LIN {X 0,Y 488.67,Z 344.234,A -85,B 0,C 180,E1 -6456.253,E2 -6456.253} C_VEL
LIN {X 0,Y 488.747,Z 344.224,A -85,B 0,C 180,E1 -6459.176,E2 -6459.176} C_VEL
LIN {X 0,Y 488.748,Z 344.228,A -85,B 0,C 180,E1 -6461.632,E2 -6461.632} C_VEL
LIN {X 0,Y 488.762,Z 344.223,A -85,B 0,C 180,E1 -6465,E2 -6465} C_VEL
LIN {X 0,Y 488.806,Z 344.211,A -85,B 0,C 180,E1 -6468.387,E2 -6468.387} C_VEL
LIN {X 0,Y 488.786,Z 344.226,A -85,B 0,C 180,E1 -6471.733,E2 -6471.733} C_VEL
LIN {X 0,Y 488.853,Z 344.206,A -85,B 0,C 180,E1 -6474.224,E2 -6474.224} C_VEL
LIN {X 0,Y 488.953,Z 344.207,A -85,B 0,C 180,E1 -6477.529,E2 -6477.529} C_VEL
LIN {X 0,Y 488.97,Z 344.194,A -85,B 0,C 180,E1 -6480,E2 -6480} C_VEL
LIN {X 0,Y 488.956,Z 344.194,A -85,B 0,C 180,E1 -6482.471,E2 -6482.471} C_VEL
LIN {X 0,Y 488.842,Z 344.213,A -85,B 0,C 180,E1 -6485.776,E2 -6485.776} C_VEL
LIN {X 0,Y 488.787,Z 344.212,A -85,B 0,C 180,E1 -6488.267,E2 -6488.267} C_VEL
LIN {X 0,Y 488.806,Z 344.219,A -85,B 0,C 180,E1 -6491.612,E2 -6491.612} C_VEL
LIN {X 0,Y 488.762,Z 344.22,A -85,B 0,C 180,E1 -6495,E2 -6495} C_VEL
LIN {X 0,Y 488.747,Z 344.223,A -85,B 0,C 180,E1 -6498.442,E2 -6498.442} C_VEL
LIN {X 0,Y 488.707,Z 344.231,A -85,B 0,C 180,E1 -6501.071,E2 -6501.071} C_VEL
LIN {X 0,Y 488.684,Z 344.231,A -85,B 0,C 180,E1 -6503.746,E2 -6503.746} C_VEL
LIN {X 0,Y 488.792,Z 344.223,A -85,B 0,C 180,E1 -6506.944,E2 -6506.944} C_VEL
LIN {X 0,Y 488.71,Z 344.225,A -85,B 0,C 180,E1 -6510.363,E2 -6510.363} C_VEL
LIN {X 0,Y 488.734,Z 344.226,A -85,B 0,C 180,E1 -6513.484,E2 -6513.484} C_VEL
LIN {X 0,Y 488.682,Z 344.235,A -85,B 0,C 180,E1 -6516.354,E2 -6516.354} C_VEL
LIN {X 0,Y 488.701,Z 344.217,A -85,B 0,C 180,E1 -6519.254,E2 -6519.254} C_VEL
LIN {X 0,Y 488.709,Z 344.228,A -85,B 0,C 180,E1 -6521.6,E2 -6521.6} C_VEL
LIN {X 0,Y 488.712,Z 344.234,A -85,B 0,C 180,E1 -6524.801,E2 -6524.801} C_VEL
LIN {X 0,Y 488.692,Z 344.227,A -85,B 0,C 180,E1 -6527.475,E2 -6527.475} C_VEL
LIN {X 0,Y 488.733,Z 344.229,A -85,B 0,C 180,E1 -6529.677,E2 -6529.677} C_VEL
LIN {X 0,Y 488.68,Z 344.241,A -85,B 0,C 180,E1 -6532.841,E2 -6532.841} C_VEL
LIN {X 0,Y 488.73,Z 344.231,A -85,B 0,C 180,E1 -6535.887,E2 -6535.887} C_VEL
LIN {X 0,Y 488.692,Z 344.238,A -85,B 0,C 180,E1 -6538.82,E2 -6538.82} C_VEL
LIN {X 0,Y 488.769,Z 344.487,A -85,B 0,C 180,E1 -6540.052,E2 -6540.052} C_VEL
LIN {X 0,Y 493.274,Z 361.433,A -85,B 0,C 180,E1 -6542.558,E2 -6542.558} C_VEL
LIN {X 0,Y 493.811,Z 363.917,A -85,B 0,C 180,E1 -6542.907,E2 -6542.907} C_VEL
LIN {X 0,Y 492.75,Z 385.348,A -85,B 0,C 180,E1 -6545.568,E2 -6545.568} C_VEL
LIN {X 0,Y 492.176,Z 397.96,A -85,B 0,C 180,E1 -6547.086,E2 -6547.086} C_VEL
LIN {X 0,Y 493.705,Z 407.128,A -85,B 0,C 180,E1 -6547.34,E2 -6547.34} C_VEL
LIN {X 0,Y 495.118,Z 416.237,A -85,B 0,C 180,E1 -6547.557,E2 -6547.557} C_VEL
LIN {X 0,Y 493.738,Z 536.271,A -85,B 0,C 180,E1 -6549.427,E2 -6549.427} C_VEL
LIN {X 0,Y 493.419,Z 566.389,A -85,B 0,C 180,E1 -6549.902,E2 -6549.902} C_VEL
LIN {X 0,Y 493.068,Z 581.521,A -85,B 0,C 180,E1 -6550.306,E2 -6550.306} C_VEL
LIN {X 0,Y 492.614,Z 595.743,A -85,B 0,C 180,E1 -6550.844,E2 -6550.844} C_VEL
LIN {X 0,Y 491.977,Z 610.35,A -85,B 0,C 180,E1 -6551.575,E2 -6551.575} C_VEL
LIN {X 0,Y 491.358,Z 623.614,A -85,B 0,C 180,E1 -6552.413,E2 -6552.413} C_VEL
LIN {X 0,Y 490.716,Z 636.907,A -85,B 0,C 180,E1 -6553.447,E2 -6553.447} C_VEL
LIN {X 0,Y 490.068,Z 649.271,A -85,B 0,C 180,E1 -6554.615,E2 -6554.615} C_VEL
LIN {X 0,Y 489.488,Z 660.375,A -85,B 0,C 180,E1 -6555.872,E2 -6555.872} C_VEL
LIN {X 0,Y 488.978,Z 671.128,A -85,B 0,C 180,E1 -6557.339,E2 -6557.339} C_VEL
LIN {X 0,Y 488.576,Z 680.063,A -85,B 0,C 180,E1 -6558.803,E2 -6558.803} C_VEL
LIN {X 0,Y 488.296,Z 686.584,A -85,B 0,C 180,E1 -6560.054,E2 -6560.054} C_VEL
LIN {X 0,Y 488.131,Z 693.802,A -85,B 0,C 180,E1 -6561.722,E2 -6561.722} C_VEL
LIN {X 0,Y 487.997,Z 699.465,A -85,B 0,C 180,E1 -6563.384,E2 -6563.384} C_VEL
LIN {X 0,Y 487.928,Z 703.738,A -85,B 0,C 180,E1 -6565.042,E2 -6565.042} C_VEL
LIN {X 0,Y 487.946,Z 706.729,A -85,B 0,C 180,E1 -6566.697,E2 -6566.697} C_VEL
LIN {X 0,Y 487.889,Z 708.505,A -85,B 0,C 180,E1 -6568.349,E2 -6568.349} C_VEL
LIN {X 0,Y 487.816,Z 709.096,A -85,B 0,C 180,E1 -6570,E2 -6570} C_VEL
LIN {X 0,Y 487.89,Z 708.466,A -85,B 0,C 180,E1 -6571.651,E2 -6571.651} C_VEL
LIN {X 0,Y 487.947,Z 706.652,A -85,B 0,C 180,E1 -6573.303,E2 -6573.303} C_VEL
LIN {X 0,Y 487.927,Z 703.612,A -85,B 0,C 180,E1 -6574.958,E2 -6574.958} C_VEL
LIN {X 0,Y 487.992,Z 699.278,A -85,B 0,C 180,E1 -6576.616,E2 -6576.616} C_VEL
LIN {X 0,Y 488.131,Z 693.56,A -85,B 0,C 180,E1 -6578.278,E2 -6578.278} C_VEL
LIN {X 0,Y 488.294,Z 686.458,A -85,B 0,C 180,E1 -6579.946,E2 -6579.946} C_VEL
LIN {X 0,Y 488.641,Z 678.867,A -85,B 0,C 180,E1 -6581.406,E2 -6581.406} C_VEL
LIN {X 0,Y 489.055,Z 669.708,A -85,B 0,C 180,E1 -6582.87,E2 -6582.87} C_VEL
LIN {X 0,Y 489.498,Z 660.375,A -85,B 0,C 180,E1 -6584.128,E2 -6584.128} C_VEL
LIN {X 0,Y 490.044,Z 649.264,A -85,B 0,C 180,E1 -6585.386,E2 -6585.386} C_VEL
LIN {X 0,Y 490.741,Z 636.855,A -85,B 0,C 180,E1 -6586.556,E2 -6586.556} C_VEL
LIN {X 0,Y 491.377,Z 623.612,A -85,B 0,C 180,E1 -6587.587,E2 -6587.587} C_VEL
LIN {X 0,Y 491.994,Z 610.353,A -85,B 0,C 180,E1 -6588.424,E2 -6588.424} C_VEL
LIN {X 0,Y 492.62,Z 595.727,A -85,B 0,C 180,E1 -6589.156,E2 -6589.156} C_VEL
LIN {X 0,Y 493.109,Z 580.58,A -85,B 0,C 180,E1 -6589.725,E2 -6589.725} C_VEL
LIN {X 0,Y 493.458,Z 565.175,A -85,B 0,C 180,E1 -6590.123,E2 -6590.123} C_VEL
LIN {X 0,Y 494.855,Z 418.053,A -85,B 0,C 180,E1 -6592.352,E2 -6592.352} C_VEL
LIN {X 0,Y 494.694,Z 413.968,A -85,B 0,C 180,E1 -6592.433,E2 -6592.433} C_VEL
LIN {X 0,Y 492.106,Z 398.162,A -85,B 0,C 180,E1 -6592.861,E2 -6592.861} C_VEL
LIN {X 0,Y 493.384,Z 375.124,A -85,B 0,C 180,E1 -6595.737,E2 -6595.737} C_VEL
LIN {X 0,Y 494.102,Z 364.814,A -85,B 0,C 180,E1 -6597.075,E2 -6597.075} C_VEL
LIN {X 0,Y 491.36,Z 353.308,A -85,B 0,C 180,E1 -6598.888,E2 -6598.888} C_VEL
LIN {X 0,Y 488.742,Z 344.352,A -85,B 0,C 180,E1 -6600.478,E2 -6600.478} C_VEL
LIN {X 0,Y 488.736,Z 344.232,A -85,B 0,C 180,E1 -6603.484,E2 -6603.484} C_VEL
LIN {X 0,Y 488.685,Z 344.239,A -85,B 0,C 180,E1 -6606.355,E2 -6606.355} C_VEL
LIN {X 0,Y 488.702,Z 344.238,A -85,B 0,C 180,E1 -6609.254,E2 -6609.254} C_VEL
LIN {X 0,Y 488.707,Z 344.233,A -85,B 0,C 180,E1 -6611.6,E2 -6611.6} C_VEL
LIN {X 0,Y 488.702,Z 344.239,A -85,B 0,C 180,E1 -6614.803,E2 -6614.803} C_VEL
LIN {X 0,Y 488.689,Z 344.236,A -85,B 0,C 180,E1 -6617.474,E2 -6617.474} C_VEL
LIN {X 0,Y 488.701,Z 344.238,A -85,B 0,C 180,E1 -6620.746,E2 -6620.746} C_VEL
LIN {X 0,Y 488.67,Z 344.241,A -85,B 0,C 180,E1 -6623.867,E2 -6623.867} C_VEL
LIN {X 0,Y 488.737,Z 344.233,A -85,B 0,C 180,E1 -6626.877,E2 -6626.877} C_VEL
LIN {X 0,Y 488.719,Z 344.236,A -85,B 0,C 180,E1 -6629.78,E2 -6629.78} C_VEL
LIN {X 0,Y 488.736,Z 344.505,A -85,B 0,C 180,E1 -6631.148,E2 -6631.148} C_VEL
LIN {X 0,Y 491.865,Z 356.433,A -85,B 0,C 180,E1 -6633.48,E2 -6633.48} C_VEL
LIN {X 0,Y 493.058,Z 363.175,A -85,B 0,C 180,E1 -6634.684,E2 -6634.684} C_VEL
LIN {X 0,Y 491.663,Z 386.383,A -85,B 0,C 180,E1 -6638.3,E2 -6638.3} C_VEL
LIN {X 0,Y 491.166,Z 398.04,A -85,B 0,C 180,E1 -6640.038,E2 -6640.038} C_VEL
LIN {X 0,Y 494.175,Z 414.23,A -85,B 0,C 180,E1 -6640.519,E2 -6640.519} C_VEL
LIN {X 0,Y 492.63,Z 511.877,A -85,B 0,C 180,E1 -6642.219,E2 -6642.219} C_VEL
LIN {X 0,Y 492.189,Z 540.322,A -85,B 0,C 180,E1 -6642.728,E2 -6642.728} C_VEL
LIN {X 0,Y 491.852,Z 554.764,A -85,B 0,C 180,E1 -6643.155,E2 -6643.155} C_VEL
LIN {X 0,Y 491.483,Z 569.057,A -85,B 0,C 180,E1 -6643.756,E2 -6643.756} C_VEL
LIN {X 0,Y 491.035,Z 581.402,A -85,B 0,C 180,E1 -6644.433,E2 -6644.433} C_VEL
LIN {X 0,Y 490.524,Z 593.611,A -85,B 0,C 180,E1 -6645.267,E2 -6645.267} C_VEL
LIN {X 0,Y 490.005,Z 605.948,A -85,B 0,C 180,E1 -6646.311,E2 -6646.311} C_VEL
LIN {X 0,Y 489.55,Z 616.291,A -85,B 0,C 180,E1 -6647.375,E2 -6647.375} C_VEL
LIN {X 0,Y 489.153,Z 626.192,A -85,B 0,C 180,E1 -6648.606,E2 -6648.606} C_VEL
LIN {X 0,Y 488.76,Z 634.535,A -85,B 0,C 180,E1 -6649.855,E2 -6649.855} C_VEL
LIN {X 0,Y 488.47,Z 642.486,A -85,B 0,C 180,E1 -6651.311,E2 -6651.311} C_VEL
LIN {X 0,Y 488.253,Z 648.047,A -85,B 0,C 180,E1 -6652.557,E2 -6652.557} C_VEL
LIN {X 0,Y 488.163,Z 653.848,A -85,B 0,C 180,E1 -6654.216,E2 -6654.216} C_VEL
LIN {X 0,Y 487.974,Z 656.147,A -85,B 0,C 180,E1 -6655.043,E2 -6655.043} C_VEL
LIN {X 0,Y 488.064,Z 658.053,A -85,B 0,C 180,E1 -6655.871,E2 -6655.871} C_VEL
LIN {X 0,Y 487.987,Z 660.799,A -85,B 0,C 180,E1 -6657.524,E2 -6657.524} C_VEL
LIN {X 0,Y 487.831,Z 662.169,A -85,B 0,C 180,E1 -6659.175,E2 -6659.175} C_VEL
LIN {X 0,Y 487.831,Z 662.181,A -85,B 0,C 180,E1 -6660.826,E2 -6660.826} C_VEL
LIN {X 0,Y 487.987,Z 660.829,A -85,B 0,C 180,E1 -6662.476,E2 -6662.476} C_VEL
LIN {X 0,Y 488.043,Z 658.097,A -85,B 0,C 180,E1 -6664.129,E2 -6664.129} C_VEL
LIN {X 0,Y 488.06,Z 655.112,A -85,B 0,C 180,E1 -6665.371,E2 -6665.371} C_VEL
LIN {X 0,Y 488.144,Z 651.07,A -85,B 0,C 180,E1 -6666.663,E2 -6666.663} C_VEL
LIN {X 0,Y 488.36,Z 644.627,A -85,B 0,C 180,E1 -6668.274,E2 -6668.274} C_VEL
LIN {X 0,Y 488.647,Z 637.248,A -85,B 0,C 180,E1 -6669.73,E2 -6669.73} C_VEL
LIN {X 0,Y 489.05,Z 628.073,A -85,B 0,C 180,E1 -6671.187,E2 -6671.187} C_VEL
LIN {X 0,Y 489.464,Z 618.122,A -85,B 0,C 180,E1 -6672.476,E2 -6672.476} C_VEL
LIN {X 0,Y 489.886,Z 607.773,A -85,B 0,C 180,E1 -6673.587,E2 -6673.587} C_VEL
LIN {X 0,Y 490.398,Z 595.975,A -85,B 0,C 180,E1 -6674.631,E2 -6674.631} C_VEL
LIN {X 0,Y 490.984,Z 582.874,A -85,B 0,C 180,E1 -6675.569,E2 -6675.569} C_VEL
LIN {X 0,Y 491.461,Z 570.021,A -85,B 0,C 180,E1 -6676.299,E2 -6676.299} C_VEL
LIN {X 0,Y 491.859,Z 555.768,A -85,B 0,C 180,E1 -6676.918,E2 -6676.918} C_VEL
LIN {X 0,Y 492.294,Z 541.273,A -85,B 0,C 180,E1 -6677.357,E2 -6677.357} C_VEL
LIN {X 0,Y 492.476,Z 525.847,A -85,B 0,C 180,E1 -6677.653,E2 -6677.653} C_VEL
LIN {X 0,Y 493.822,Z 414.339,A -85,B 0,C 180,E1 -6679.448,E2 -6679.448} C_VEL
LIN {X 0,Y 490.808,Z 397.758,A -85,B 0,C 180,E1 -6679.875,E2 -6679.875} C_VEL
LIN {X 0,Y 491.591,Z 378.455,A -85,B 0,C 180,E1 -6682.706,E2 -6682.706} C_VEL
LIN {X 0,Y 492.374,Z 360.916,A -85,B 0,C 180,E1 -6685.354,E2 -6685.354} C_VEL
LIN {X 0,Y 490.258,Z 350.903,A -85,B 0,C 180,E1 -6687.034,E2 -6687.034} C_VEL
LIN {X 0,Y 488.753,Z 344.554,A -85,B 0,C 180,E1 -6688.153,E2 -6688.153} C_VEL
LIN {X 0,Y 488.695,Z 344.246,A -85,B 0,C 180,E1 -6688.332,E2 -6688.332} C_VEL
LIN {X 0,Y 488.659,Z 344.24,A -85,B 0,C 180,E1 -6691.182,E2 -6691.182} C_VEL
LIN {X 0,Y 488.703,Z 344.239,A -85,B 0,C 180,E1 -6694.115,E2 -6694.115} C_VEL
LIN {X 0,Y 488.646,Z 344.24,A -85,B 0,C 180,E1 -6697.162,E2 -6697.162} C_VEL
LIN {X 0,Y 488.668,Z 344.24,A -85,B 0,C 180,E1 -6700.33,E2 -6700.33} C_VEL
LIN {X 0,Y 488.658,Z 344.232,A -85,B 0,C 180,E1 -6703.562,E2 -6703.562} C_VEL
LIN {X 0,Y 488.027,Z 344.322,A -85,B 0,C 180,E1 -6704.249,E2 -6704.249} C_VEL
LIN {X 0,Y 485.175,Z 344.673,A -85,B 0,C 180,E1 -6705.366,E2 -6705.366} C_VEL
LIN {X 0,Y 482.736,Z 344.972,A -85,B 0,C 180,E1 -6706.266,E2 -6706.266} C_VEL
LIN {X 0,Y 481.682,Z 345.099,A -85,B 0,C 180,E1 -6706.962,E2 -6706.962} C_VEL
LIN {X 0,Y 481.595,Z 345.11,A -85,B 0,C 180,E1 -6707.197,E2 -6707.197} C_VEL
LIN {X 0,Y 481.628,Z 345.113,A -85,B 0,C 180,E1 -6710.055,E2 -6710.055} C_VEL
LIN {X 0,Y 481.603,Z 345.114,A -85,B 0,C 180,E1 -6713.251,E2 -6713.251} C_VEL
LIN {X 0,Y 481.671,Z 345.113,A -85,B 0,C 180,E1 -6716.327,E2 -6716.327} C_VEL
LIN {X 0,Y 481.632,Z 345.309,A -85,B 0,C 180,E1 -6719.478,E2 -6719.478} C_VEL
LIN {X 0,Y 485.46,Z 360.506,A -85,B 0,C 180,E1 -6721.798,E2 -6721.798} C_VEL
LIN {X 0,Y 486.304,Z 365.031,A -85,B 0,C 180,E1 -6722.454,E2 -6722.454} C_VEL
LIN {X 0,Y 485.411,Z 387.512,A -85,B 0,C 180,E1 -6725.385,E2 -6725.385} C_VEL
LIN {X 0,Y 485.132,Z 397.848,A -85,B 0,C 180,E1 -6726.645,E2 -6726.645} C_VEL
LIN {X 0,Y 488.991,Z 418.099,A -85,B 0,C 180,E1 -6727.166,E2 -6727.166} C_VEL
LIN {X 0,Y 487.489,Z 565.061,A -85,B 0,C 180,E1 -6729.407,E2 -6729.407} C_VEL
LIN {X 0,Y 487.064,Z 580.106,A -85,B 0,C 180,E1 -6729.794,E2 -6729.794} C_VEL
LIN {X 0,Y 486.479,Z 595.122,A -85,B 0,C 180,E1 -6730.351,E2 -6730.351} C_VEL
LIN {X 0,Y 485.866,Z 608.495,A -85,B 0,C 180,E1 -6731.006,E2 -6731.006} C_VEL
LIN {X 0,Y 485.213,Z 622.242,A -85,B 0,C 180,E1 -6731.855,E2 -6731.855} C_VEL
LIN {X 0,Y 484.433,Z 634.862,A -85,B 0,C 180,E1 -6732.807,E2 -6732.807} C_VEL
LIN {X 0,Y 483.707,Z 647.615,A -85,B 0,C 180,E1 -6733.975,E2 -6733.975} C_VEL
LIN {X 0,Y 483.081,Z 657.437,A -85,B 0,C 180,E1 -6735.035,E2 -6735.035} C_VEL
LIN {X 0,Y 482.49,Z 667.455,A -85,B 0,C 180,E1 -6736.308,E2 -6736.308} C_VEL
LIN {X 0,Y 481.889,Z 677.81,A -85,B 0,C 180,E1 -6737.888,E2 -6737.888} C_VEL
LIN {X 0,Y 481.597,Z 685.38,A -85,B 0,C 180,E1 -6739.277,E2 -6739.277} C_VEL
LIN {X 0,Y 481.239,Z 692.115,A -85,B 0,C 180,E1 -6740.756,E2 -6740.756} C_VEL
LIN {X 0,Y 481.016,Z 698.355,A -85,B 0,C 180,E1 -6742.444,E2 -6742.444} C_VEL
LIN {X 0,Y 480.915,Z 703.186,A -85,B 0,C 180,E1 -6744.128,E2 -6744.128} C_VEL
LIN {X 0,Y 480.796,Z 706.733,A -85,B 0,C 180,E1 -6745.809,E2 -6745.809} C_VEL
LIN {X 0,Y 480.8,Z 709.075,A -85,B 0,C 180,E1 -6747.487,E2 -6747.487} C_VEL
LIN {X 0,Y 480.757,Z 710.268,A -85,B 0,C 180,E1 -6749.162,E2 -6749.162} C_VEL
LIN {X 0,Y 480.757,Z 710.285,A -85,B 0,C 180,E1 -6750.838,E2 -6750.838} C_VEL
LIN {X 0,Y 480.8,Z 709.156,A -85,B 0,C 180,E1 -6752.513,E2 -6752.513} C_VEL
LIN {X 0,Y 480.796,Z 706.883,A -85,B 0,C 180,E1 -6754.191,E2 -6754.191} C_VEL
LIN {X 0,Y 480.921,Z 703.413,A -85,B 0,C 180,E1 -6755.871,E2 -6755.871} C_VEL
LIN {X 0,Y 481.009,Z 698.658,A -85,B 0,C 180,E1 -6757.556,E2 -6757.556} C_VEL
LIN {X 0,Y 481.219,Z 692.491,A -85,B 0,C 180,E1 -6759.245,E2 -6759.245} C_VEL
LIN {X 0,Y 481.617,Z 684.74,A -85,B 0,C 180,E1 -6760.935,E2 -6760.935} C_VEL
LIN {X 0,Y 482.001,Z 676.224,A -85,B 0,C 180,E1 -6762.461,E2 -6762.461} C_VEL
LIN {X 0,Y 482.563,Z 666.53,A -85,B 0,C 180,E1 -6763.904,E2 -6763.904} C_VEL
LIN {X 0,Y 483.131,Z 656.375,A -85,B 0,C 180,E1 -6765.179,E2 -6765.179} C_VEL
LIN {X 0,Y 483.861,Z 644.214,A -85,B 0,C 180,E1 -6766.454,E2 -6766.454} C_VEL
LIN {X 0,Y 484.626,Z 632.086,A -85,B 0,C 180,E1 -6767.512,E2 -6767.512} C_VEL
LIN {X 0,Y 485.389,Z 618.859,A -85,B 0,C 180,E1 -6768.465,E2 -6768.465} C_VEL
LIN {X 0,Y 486.055,Z 605.273,A -85,B 0,C 180,E1 -6769.26,E2 -6769.26} C_VEL
LIN {X 0,Y 486.718,Z 589.87,A -85,B 0,C 180,E1 -6769.958,E2 -6769.958} C_VEL
LIN {X 0,Y 487.207,Z 575.123,A -85,B 0,C 180,E1 -6770.448,E2 -6770.448} C_VEL
LIN {X 0,Y 487.572,Z 559.443,A -85,B 0,C 180,E1 -6770.79,E2 -6770.79} C_VEL
LIN {X 0,Y 488.93,Z 417.561,A -85,B 0,C 180,E1 -6772.936,E2 -6772.936} C_VEL
LIN {X 0,Y 485.145,Z 397.66,A -85,B 0,C 180,E1 -6773.458,E2 -6773.458} C_VEL
LIN {X 0,Y 485.658,Z 381.364,A -85,B 0,C 180,E1 -6775.5,E2 -6775.5} C_VEL
LIN {X 0,Y 486.267,Z 364.634,A -85,B 0,C 180,E1 -6777.698,E2 -6777.698} C_VEL
LIN {X 0,Y 483.266,Z 351.613,A -85,B 0,C 180,E1 -6779.634,E2 -6779.634} C_VEL
LIN {X 0,Y 481.645,Z 345.259,A -85,B 0,C 180,E1 -6780.631,E2 -6780.631} C_VEL
LIN {X 0,Y 481.649,Z 345.109,A -85,B 0,C 180,E1 -6783.724,E2 -6783.724} C_VEL
LIN {X 0,Y 481.602,Z 345.118,A -85,B 0,C 180,E1 -6786.749,E2 -6786.749} C_VEL
LIN {X 0,Y 481.627,Z 345.11,A -85,B 0,C 180,E1 -6789.945,E2 -6789.945} C_VEL
LIN {X 0,Y 481.618,Z 345.115,A -85,B 0,C 180,E1 -6793.302,E2 -6793.302} C_VEL
LIN {X 0,Y 481.652,Z 345.113,A -85,B 0,C 180,E1 -6795.642,E2 -6795.642} C_VEL
LIN {X 0,Y 481.62,Z 345.115,A -85,B 0,C 180,E1 -6798.954,E2 -6798.954} C_VEL
LIN {X 0,Y 481.633,Z 345.119,A -85,B 0,C 180,E1 -6801.996,E2 -6801.996} C_VEL
LIN {X 0,Y 481.68,Z 345.105,A -85,B 0,C 180,E1 -6805.317,E2 -6805.317} C_VEL
LIN {X 0,Y 481.643,Z 345.107,A -85,B 0,C 180,E1 -6808.311,E2 -6808.311} C_VEL
LIN {X 0,Y 481.673,Z 345.11,A -85,B 0,C 180,E1 -6811.217,E2 -6811.217} C_VEL
LIN {X 0,Y 481.643,Z 345.114,A -85,B 0,C 180,E1 -6814.039,E2 -6814.039} C_VEL
LIN {X 0,Y 481.675,Z 345.105,A -85,B 0,C 180,E1 -6816.812,E2 -6816.812} C_VEL
LIN {X 0,Y 481.696,Z 345.107,A -85,B 0,C 180,E1 -6819.503,E2 -6819.503} C_VEL
LIN {X 0,Y 481.689,Z 345.101,A -85,B 0,C 180,E1 -6822.158,E2 -6822.158} C_VEL
LIN {X 0,Y 481.743,Z 345.096,A -85,B 0,C 180,E1 -6824.776,E2 -6824.776} C_VEL
LIN {X 0,Y 481.752,Z 345.091,A -85,B 0,C 180,E1 -6828.215,E2 -6828.215} C_VEL
LIN {X 0,Y 481.74,Z 345.105,A -85,B 0,C 180,E1 -6831.611,E2 -6831.611} C_VEL
LIN {X 0,Y 481.814,Z 345.083,A -85,B 0,C 180,E1 -6834.139,E2 -6834.139} C_VEL
LIN {X 0,Y 481.919,Z 345.082,A -85,B 0,C 180,E1 -6837.492,E2 -6837.492} C_VEL
LIN {X 0,Y 481.941,Z 345.07,A -85,B 0,C 180,E1 -6840,E2 -6840} C_VEL
LIN {X 0,Y 481.922,Z 345.07,A -85,B 0,C 180,E1 -6842.507,E2 -6842.507} C_VEL
LIN {X 0,Y 481.801,Z 345.089,A -85,B 0,C 180,E1 -6845.861,E2 -6845.861} C_VEL
LIN {X 0,Y 481.741,Z 345.09,A -85,B 0,C 180,E1 -6848.389,E2 -6848.389} C_VEL
LIN {X 0,Y 481.752,Z 345.096,A -85,B 0,C 180,E1 -6851.785,E2 -6851.785} C_VEL
LIN {X 0,Y 481.743,Z 345.098,A -85,B 0,C 180,E1 -6855.224,E2 -6855.224} C_VEL
LIN {X 0,Y 481.709,Z 345.101,A -85,B 0,C 180,E1 -6858.722,E2 -6858.722} C_VEL
LIN {X 0,Y 481.647,Z 345.116,A -85,B 0,C 180,E1 -6861.395,E2 -6861.395} C_VEL
LIN {X 0,Y 481.67,Z 345.103,A -85,B 0,C 180,E1 -6864.113,E2 -6864.113} C_VEL
LIN {X 0,Y 481.747,Z 345.104,A -85,B 0,C 180,E1 -6867.139,E2 -6867.139} C_VEL
LIN {X 0,Y 481.679,Z 345.101,A -85,B 0,C 180,E1 -6869.741,E2 -6869.741} C_VEL
LIN {X 0,Y 481.672,Z 345.111,A -85,B 0,C 180,E1 -6872.674,E2 -6872.674} C_VEL
LIN {X 0,Y 481.637,Z 345.113,A -85,B 0,C 180,E1 -6875.709,E2 -6875.709} C_VEL
LIN {X 0,Y 481.671,Z 345.099,A -85,B 0,C 180,E1 -6878.859,E2 -6878.859} C_VEL
LIN {X 0,Y 481.654,Z 345.105,A -85,B 0,C 180,E1 -6881.913,E2 -6881.913} C_VEL
LIN {X 0,Y 481.66,Z 345.112,A -85,B 0,C 180,E1 -6884.457,E2 -6884.457} C_VEL
LIN {X 0,Y 481.648,Z 345.105,A -85,B 0,C 180,E1 -6887.839,E2 -6887.839} C_VEL
LIN {X 0,Y 481.681,Z 345.111,A -85,B 0,C 180,E1 -6890.651,E2 -6890.651} C_VEL
LIN {X 0,Y 481.627,Z 345.116,A -85,B 0,C 180,E1 -6893.376,E2 -6893.376} C_VEL
LIN {X 0,Y 481.71,Z 345.108,A -85,B 0,C 180,E1 -6896.33,E2 -6896.33} C_VEL
LIN {X 0,Y 481.72,Z 345.277,A -85,B 0,C 180,E1 -6899.69,E2 -6899.69} C_VEL
LIN {X 0,Y 486.112,Z 361.759,A -85,B 0,C 180,E1 -6902.185,E2 -6902.185} C_VEL
LIN {X 0,Y 486.996,Z 365.544,A -85,B 0,C 180,E1 -6902.729,E2 -6902.729} C_VEL
LIN {X 0,Y 486.309,Z 379.817,A -85,B 0,C 180,E1 -6904.536,E2 -6904.536} C_VEL
LIN {X 0,Y 485.379,Z 397.859,A -85,B 0,C 180,E1 -6906.761,E2 -6906.761} C_VEL
LIN {X 0,Y 486.072,Z 402.084,A -85,B 0,C 180,E1 -6906.908,E2 -6906.908} C_VEL
LIN {X 0,Y 488.492,Z 417.195,A -85,B 0,C 180,E1 -6907.274,E2 -6907.274} C_VEL
LIN {X 0,Y 487.464,Z 502.409,A -85,B 0,C 180,E1 -6908.624,E2 -6908.624} C_VEL
LIN {X 0,Y 486.823,Z 565.34,A -85,B 0,C 180,E1 -6909.59,E2 -6909.59} C_VEL
LIN {X 0,Y 486.403,Z 581.053,A -85,B 0,C 180,E1 -6910.004,E2 -6910.004} C_VEL
LIN {X 0,Y 485.904,Z 595.807,A -85,B 0,C 180,E1 -6910.569,E2 -6910.569} C_VEL
LIN {X 0,Y 485.218,Z 610.4,A -85,B 0,C 180,E1 -6911.309,E2 -6911.309} C_VEL
LIN {X 0,Y 484.563,Z 623.657,A -85,B 0,C 180,E1 -6912.158,E2 -6912.158} C_VEL
LIN {X 0,Y 483.853,Z 637.104,A -85,B 0,C 180,E1 -6913.22,E2 -6913.22} C_VEL
LIN {X 0,Y 483.156,Z 649.303,A -85,B 0,C 180,E1 -6914.389,E2 -6914.389} C_VEL
LIN {X 0,Y 482.537,Z 660.403,A -85,B 0,C 180,E1 -6915.665,E2 -6915.665} C_VEL
LIN {X 0,Y 481.997,Z 671.152,A -85,B 0,C 180,E1 -6917.152,E2 -6917.152} C_VEL
LIN {X 0,Y 481.565,Z 680.074,A -85,B 0,C 180,E1 -6918.637,E2 -6918.637} C_VEL
LIN {X 0,Y 481.257,Z 686.473,A -85,B 0,C 180,E1 -6919.907,E2 -6919.907} C_VEL
LIN {X 0,Y 481.057,Z 693.547,A -85,B 0,C 180,E1 -6921.599,E2 -6921.599} C_VEL
LIN {X 0,Y 480.908,Z 699.113,A -85,B 0,C 180,E1 -6923.286,E2 -6923.286} C_VEL
LIN {X 0,Y 480.854,Z 703.387,A -85,B 0,C 180,E1 -6924.969,E2 -6924.969} C_VEL
LIN {X 0,Y 480.87,Z 706.389,A -85,B 0,C 180,E1 -6926.649,E2 -6926.649} C_VEL
LIN {X 0,Y 480.82,Z 708.17,A -85,B 0,C 180,E1 -6928.325,E2 -6928.325} C_VEL
LIN {X 0,Y 480.74,Z 708.76,A -85,B 0,C 180,E1 -6930,E2 -6930} C_VEL
LIN {X 0,Y 480.821,Z 708.122,A -85,B 0,C 180,E1 -6931.675,E2 -6931.675} C_VEL
LIN {X 0,Y 480.87,Z 706.291,A -85,B 0,C 180,E1 -6933.352,E2 -6933.352} C_VEL
LIN {X 0,Y 480.853,Z 703.294,A -85,B 0,C 180,E1 -6935.031,E2 -6935.031} C_VEL
LIN {X 0,Y 480.902,Z 699.097,A -85,B 0,C 180,E1 -6936.714,E2 -6936.714} C_VEL
LIN {X 0,Y 481.057,Z 693.546,A -85,B 0,C 180,E1 -6938.401,E2 -6938.401} C_VEL
LIN {X 0,Y 481.258,Z 686.478,A -85,B 0,C 180,E1 -6940.093,E2 -6940.093} C_VEL
LIN {X 0,Y 481.619,Z 678.889,A -85,B 0,C 180,E1 -6941.575,E2 -6941.575} C_VEL
LIN {X 0,Y 482.07,Z 669.733,A -85,B 0,C 180,E1 -6943.06,E2 -6943.06} C_VEL
LIN {X 0,Y 482.558,Z 660.402,A -85,B 0,C 180,E1 -6944.335,E2 -6944.335} C_VEL
LIN {X 0,Y 483.179,Z 649.295,A -85,B 0,C 180,E1 -6945.61,E2 -6945.61} C_VEL
LIN {X 0,Y 483.872,Z 637.066,A -85,B 0,C 180,E1 -6946.782,E2 -6946.782} C_VEL
LIN {X 0,Y 484.573,Z 623.653,A -85,B 0,C 180,E1 -6947.842,E2 -6947.842} C_VEL
LIN {X 0,Y 485.259,Z 610.4,A -85,B 0,C 180,E1 -6948.689,E2 -6948.689} C_VEL
LIN {X 0,Y 485.911,Z 595.785,A -85,B 0,C 180,E1 -6949.431,E2 -6949.431} C_VEL
LIN {X 0,Y 486.438,Z 580.881,A -85,B 0,C 180,E1 -6949.999,E2 -6949.999} C_VEL
LIN {X 0,Y 486.81,Z 565.304,A -85,B 0,C 180,E1 -6950.41,E2 -6950.41} C_VEL
LIN {X 0,Y 488.284,Z 416.22,A -85,B 0,C 180,E1 -6952.697,E2 -6952.697} C_VEL
LIN {X 0,Y 485.37,Z 398.056,A -85,B 0,C 180,E1 -6953.211,E2 -6953.211} C_VEL
LIN {X 0,Y 486.841,Z 374.691,A -85,B 0,C 180,E1 -6956.208,E2 -6956.208} C_VEL
LIN {X 0,Y 487.467,Z 366.922,A -85,B 0,C 180,E1 -6957.242,E2 -6957.242} C_VEL
LIN {X 0,Y 484.631,Z 355.139,A -85,B 0,C 180,E1 -6959.159,E2 -6959.159} C_VEL
LIN {X 0,Y 481.688,Z 345.226,A -85,B 0,C 180,E1 -6960.997,E2 -6960.997} C_VEL
LIN {X 0,Y 481.698,Z 345.107,A -85,B 0,C 180,E1 -6963.733,E2 -6963.733} C_VEL
LIN {X 0,Y 481.627,Z 345.12,A -85,B 0,C 180,E1 -6966.747,E2 -6966.747} C_VEL
LIN {X 0,Y 481.678,Z 345.11,A -85,B 0,C 180,E1 -6969.941,E2 -6969.941} C_VEL
LIN {X 0,Y 481.633,Z 345.117,A -85,B 0,C 180,E1 -6973.147,E2 -6973.147} C_VEL
LIN {X 0,Y 481.653,Z 345.113,A -85,B 0,C 180,E1 -6975.642,E2 -6975.642} C_VEL
LIN {X 0,Y 481.65,Z 345.115,A -85,B 0,C 180,E1 -6978.958,E2 -6978.958} C_VEL
LIN {X 0,Y 481.651,Z 345.115,A -85,B 0,C 180,E1 -6981.994,E2 -6981.994} C_VEL
LIN {X 0,Y 481.685,Z 345.11,A -85,B 0,C 180,E1 -6985.318,E2 -6985.318} C_VEL
LIN {X 0,Y 481.644,Z 345.117,A -85,B 0,C 180,E1 -6988.312,E2 -6988.312} C_VEL
LIN {X 0,Y 481.693,Z 345.301,A -85,B 0,C 180,E1 -6990.621,E2 -6990.621} C_VEL
LIN {X 0,Y 484.641,Z 356.291,A -85,B 0,C 180,E1 -6992.871,E2 -6992.871} C_VEL
LIN {X 0,Y 486.27,Z 363.898,A -85,B 0,C 180,E1 -6994.305,E2 -6994.305} C_VEL
LIN {X 0,Y 485.966,Z 370.471,A -85,B 0,C 180,E1 -6995.377,E2 -6995.377} C_VEL
LIN {X 0,Y 484.856,Z 388.641,A -85,B 0,C 180,E1 -6998.247,E2 -6998.247} C_VEL
LIN {X 0,Y 484.401,Z 398.076,A -85,B 0,C 180,E1 -6999.671,E2 -6999.671} C_VEL
LIN {X 0,Y 487.323,Z 413.098,A -85,B 0,C 180,E1 -7000.153,E2 -7000.153} C_VEL
LIN {X 0,Y 487.635,Z 415.738,A -85,B 0,C 180,E1 -7000.222,E2 -7000.222} C_VEL
LIN {X 0,Y 485.917,Z 510.801,A -85,B 0,C 180,E1 -7001.937,E2 -7001.937} C_VEL
LIN {X 0,Y 485.412,Z 540.37,A -85,B 0,C 180,E1 -7002.479,E2 -7002.479} C_VEL
LIN {X 0,Y 485.039,Z 554.787,A -85,B 0,C 180,E1 -7002.911,E2 -7002.911} C_VEL
LIN {X 0,Y 484.646,Z 569.341,A -85,B 0,C 180,E1 -7003.533,E2 -7003.533} C_VEL
LIN {X 0,Y 484.113,Z 583.163,A -85,B 0,C 180,E1 -7004.313,E2 -7004.313} C_VEL
LIN {X 0,Y 483.508,Z 596.368,A -85,B 0,C 180,E1 -7005.264,E2 -7005.264} C_VEL
LIN {X 0,Y 482.978,Z 608.246,A -85,B 0,C 180,E1 -7006.322,E2 -7006.322} C_VEL
LIN {X 0,Y 482.477,Z 618.347,A -85,B 0,C 180,E1 -7007.411,E2 -7007.411} C_VEL
LIN {X 0,Y 482.101,Z 627.89,A -85,B 0,C 180,E1 -7008.65,E2 -7008.65} C_VEL
LIN {X 0,Y 481.716,Z 636.013,A -85,B 0,C 180,E1 -7009.917,E2 -7009.917} C_VEL
LIN {X 0,Y 481.397,Z 643.771,A -85,B 0,C 180,E1 -7011.394,E2 -7011.394} C_VEL
LIN {X 0,Y 481.17,Z 649.963,A -85,B 0,C 180,E1 -7012.868,E2 -7012.868} C_VEL
LIN {X 0,Y 481.107,Z 654.164,A -85,B 0,C 180,E1 -7014.131,E2 -7014.131} C_VEL
LIN {X 0,Y 480.909,Z 656.471,A -85,B 0,C 180,E1 -7014.97,E2 -7014.97} C_VEL
LIN {X 0,Y 480.981,Z 658.386,A -85,B 0,C 180,E1 -7015.81,E2 -7015.81} C_VEL
LIN {X 0,Y 480.924,Z 661.14,A -85,B 0,C 180,E1 -7017.487,E2 -7017.487} C_VEL
LIN {X 0,Y 480.757,Z 662.513,A -85,B 0,C 180,E1 -7019.162,E2 -7019.162} C_VEL
LIN {X 0,Y 480.757,Z 662.518,A -85,B 0,C 180,E1 -7020.838,E2 -7020.838} C_VEL
LIN {X 0,Y 480.894,Z 661.153,A -85,B 0,C 180,E1 -7022.513,E2 -7022.513} C_VEL
LIN {X 0,Y 480.963,Z 658.4,A -85,B 0,C 180,E1 -7024.19,E2 -7024.19} C_VEL
LIN {X 0,Y 481.006,Z 655.393,A -85,B 0,C 180,E1 -7025.45,E2 -7025.45} C_VEL
LIN {X 0,Y 481.081,Z 651.499,A -85,B 0,C 180,E1 -7026.712,E2 -7026.712} C_VEL
LIN {X 0,Y 481.223,Z 646.686,A -85,B 0,C 180,E1 -7027.975,E2 -7027.975} C_VEL
LIN {X 0,Y 481.541,Z 639.7,A -85,B 0,C 180,E1 -7029.45,E2 -7029.45} C_VEL
LIN {X 0,Y 481.881,Z 631.023,A -85,B 0,C 180,E1 -7030.929,E2 -7030.929} C_VEL
LIN {X 0,Y 482.307,Z 622.715,A -85,B 0,C 180,E1 -7032.099,E2 -7032.099} C_VEL
LIN {X 0,Y 482.681,Z 612.931,A -85,B 0,C 180,E1 -7033.257,E2 -7033.257} C_VEL
LIN {X 0,Y 483.313,Z 600.988,A -85,B 0,C 180,E1 -7034.42,E2 -7034.42} C_VEL
LIN {X 0,Y 483.81,Z 590.443,A -85,B 0,C 180,E1 -7035.265,E2 -7035.265} C_VEL
LIN {X 0,Y 484.323,Z 577.662,A -85,B 0,C 180,E1 -7036.107,E2 -7036.107} C_VEL
LIN {X 0,Y 484.876,Z 564.173,A -85,B 0,C 180,E1 -7036.801,E2 -7036.801} C_VEL
LIN {X 0,Y 485.232,Z 549.899,A -85,B 0,C 180,E1 -7037.354,E2 -7037.354} C_VEL
LIN {X 0,Y 485.54,Z 535.76,A -85,B 0,C 180,E1 -7037.723,E2 -7037.723} C_VEL
LIN {X 0,Y 487.098,Z 415.633,A -85,B 0,C 180,E1 -7039.711,E2 -7039.711} C_VEL
LIN {X 0,Y 484.237,Z 399.511,A -85,B 0,C 180,E1 -7040.114,E2 -7040.114} C_VEL
LIN {X 0,Y 483.925,Z 397.254,A -85,B 0,C 180,E1 -7040.224,E2 -7040.224} C_VEL
LIN {X 0,Y 484.764,Z 378.494,A -85,B 0,C 180,E1 -7043.044,E2 -7043.044} C_VEL
LIN {X 0,Y 485.551,Z 363.861,A -85,B 0,C 180,E1 -7045.277,E2 -7045.277} C_VEL
LIN {X 0,Y 484.968,Z 359.206,A -85,B 0,C 180,E1 -7046.04,E2 -7046.04} C_VEL
LIN {X 0,Y 481.663,Z 345.307,A -85,B 0,C 180,E1 -7048.486,E2 -7048.486} C_VEL
LIN {X 0,Y 481.621,Z 345.12,A -85,B 0,C 180,E1 -7051.69,E2 -7051.69} C_VEL
LIN {X 0,Y 481.668,Z 345.111,A -85,B 0,C 180,E1 -7054.684,E2 -7054.684} C_VEL
LIN {X 0,Y 481.626,Z 345.12,A -85,B 0,C 180,E1 -7058.002,E2 -7058.002} C_VEL
LIN {X 0,Y 481.604,Z 345.115,A -85,B 0,C 180,E1 -7061.047,E2 -7061.047} C_VEL
LIN {X 0,Y 481.65,Z 345.114,A -85,B 0,C 180,E1 -7064.459,E2 -7064.459} C_VEL
LIN {X 0,Y 481.595,Z 345.11,A -85,B 0,C 180,E1 -7067.197,E2 -7067.197} C_VEL
LIN {X 0,Y 480.928,Z 345.201,A -85,B 0,C 180,E1 -7067.895,E2 -7067.895} C_VEL
LIN {X 0,Y 478.092,Z 345.555,A -85,B 0,C 180,E1 -7069.028,E2 -7069.028} C_VEL
LIN {X 0,Y 475.693,Z 345.853,A -85,B 0,C 180,E1 -7069.942,E2 -7069.942} C_VEL
LIN {X 0,Y 474.659,Z 345.979,A -85,B 0,C 180,E1 -7070.648,E2 -7070.648} C_VEL
LIN {X 0,Y 474.572,Z 345.989,A -85,B 0,C 180,E1 -7070.887,E2 -7070.887} C_VEL
LIN {X 0,Y 474.592,Z 345.994,A -85,B 0,C 180,E1 -7074.535,E2 -7074.535} C_VEL
LIN {X 0,Y 474.61,Z 345.989,A -85,B 0,C 180,E1 -7077.786,E2 -7077.786} C_VEL
LIN {X 0,Y 474.607,Z 346.226,A -85,B 0,C 180,E1 -7079.169,E2 -7079.169} C_VEL
LIN {X 0,Y 478.795,Z 362.833,A -85,B 0,C 180,E1 -7081.728,E2 -7081.728} C_VEL
LIN {X 0,Y 479.535,Z 366.484,A -85,B 0,C 180,E1 -7082.269,E2 -7082.269} C_VEL
LIN {X 0,Y 478.582,Z 389.263,A -85,B 0,C 180,E1 -7085.259,E2 -7085.259} C_VEL
LIN {X 0,Y 478.335,Z 397.616,A -85,B 0,C 180,E1 -7086.286,E2 -7086.286} C_VEL
LIN {X 0,Y 482.402,Z 418.761,A -85,B 0,C 180,E1 -7086.849,E2 -7086.849} C_VEL
LIN {X 0,Y 480.859,Z 564.958,A -85,B 0,C 180,E1 -7089.11,E2 -7089.11} C_VEL
LIN {X 0,Y 480.391,Z 579.836,A -85,B 0,C 180,E1 -7089.494,E2 -7089.494} C_VEL
LIN {X 0,Y 479.824,Z 594.343,A -85,B 0,C 180,E1 -7090.035,E2 -7090.035} C_VEL
LIN {X 0,Y 479.154,Z 608.457,A -85,B 0,C 180,E1 -7090.73,E2 -7090.73} C_VEL
LIN {X 0,Y 478.444,Z 622.211,A -85,B 0,C 180,E1 -7091.59,E2 -7091.59} C_VEL
LIN {X 0,Y 477.596,Z 634.835,A -85,B 0,C 180,E1 -7092.553,E2 -7092.553} C_VEL
LIN {X 0,Y 476.843,Z 647.591,A -85,B 0,C 180,E1 -7093.738,E2 -7093.738} C_VEL
LIN {X 0,Y 476.068,Z 659.165,A -85,B 0,C 180,E1 -7095.028,E2 -7095.028} C_VEL
LIN {X 0,Y 475.415,Z 668.914,A -85,B 0,C 180,E1 -7096.318,E2 -7096.318} C_VEL
LIN {X 0,Y 474.865,Z 678.295,A -85,B 0,C 180,E1 -7097.796,E2 -7097.796} C_VEL
LIN {X 0,Y 474.504,Z 686.408,A -85,B 0,C 180,E1 -7099.331,E2 -7099.331} C_VEL
LIN {X 0,Y 474.107,Z 693.816,A -85,B 0,C 180,E1 -7101.045,E2 -7101.045} C_VEL
LIN {X 0,Y 473.91,Z 699.697,A -85,B 0,C 180,E1 -7102.758,E2 -7102.758} C_VEL
LIN {X 0,Y 473.819,Z 703.172,A -85,B 0,C 180,E1 -7104.04,E2 -7104.04} C_VEL
LIN {X 0,Y 473.705,Z 706.719,A -85,B 0,C 180,E1 -7105.746,E2 -7105.746} C_VEL
LIN {X 0,Y 473.718,Z 709.062,A -85,B 0,C 180,E1 -7107.449,E2 -7107.449} C_VEL
LIN {X 0,Y 473.685,Z 710.254,A -85,B 0,C 180,E1 -7109.15,E2 -7109.15} C_VEL
LIN {X 0,Y 473.686,Z 710.271,A -85,B 0,C 180,E1 -7110.85,E2 -7110.85} C_VEL
LIN {X 0,Y 473.719,Z 709.142,A -85,B 0,C 180,E1 -7112.551,E2 -7112.551} C_VEL
LIN {X 0,Y 473.705,Z 706.867,A -85,B 0,C 180,E1 -7114.254,E2 -7114.254} C_VEL
LIN {X 0,Y 473.833,Z 703.396,A -85,B 0,C 180,E1 -7115.959,E2 -7115.959} C_VEL
LIN {X 0,Y 473.95,Z 698.639,A -85,B 0,C 180,E1 -7117.669,E2 -7117.669} C_VEL
LIN {X 0,Y 474.177,Z 692.47,A -85,B 0,C 180,E1 -7119.383,E2 -7119.383} C_VEL
LIN {X 0,Y 474.61,Z 684.716,A -85,B 0,C 180,E1 -7121.099,E2 -7121.099} C_VEL
LIN {X 0,Y 475,Z 676.472,A -85,B 0,C 180,E1 -7122.603,E2 -7122.603} C_VEL
LIN {X 0,Y 475.617,Z 666.5,A -85,B 0,C 180,E1 -7124.112,E2 -7124.112} C_VEL
LIN {X 0,Y 476.212,Z 656.343,A -85,B 0,C 180,E1 -7125.405,E2 -7125.405} C_VEL
LIN {X 0,Y 476.954,Z 644.953,A -85,B 0,C 180,E1 -7126.625,E2 -7126.625} C_VEL
LIN {X 0,Y 477.815,Z 632.045,A -85,B 0,C 180,E1 -7127.77,E2 -7127.77} C_VEL
LIN {X 0,Y 478.64,Z 618.811,A -85,B 0,C 180,E1 -7128.735,E2 -7128.735} C_VEL
LIN {X 0,Y 479.339,Z 605.215,A -85,B 0,C 180,E1 -7129.54,E2 -7129.54} C_VEL
LIN {X 0,Y 480.021,Z 590.423,A -85,B 0,C 180,E1 -7130.223,E2 -7130.223} C_VEL
LIN {X 0,Y 480.529,Z 575.972,A -85,B 0,C 180,E1 -7130.717,E2 -7130.717} C_VEL
LIN {X 0,Y 480.908,Z 560.833,A -85,B 0,C 180,E1 -7131.064,E2 -7131.064} C_VEL
LIN {X 0,Y 482.401,Z 418.704,A -85,B 0,C 180,E1 -7133.244,E2 -7133.244} C_VEL
LIN {X 0,Y 478.364,Z 397.621,A -85,B 0,C 180,E1 -7133.806,E2 -7133.806} C_VEL
LIN {X 0,Y 478.922,Z 381.158,A -85,B 0,C 180,E1 -7135.885,E2 -7135.885} C_VEL
LIN {X 0,Y 479.507,Z 367.19,A -85,B 0,C 180,E1 -7137.733,E2 -7137.733} C_VEL
LIN {X 0,Y 478.1,Z 359.965,A -85,B 0,C 180,E1 -7138.801,E2 -7138.801} C_VEL
LIN {X 0,Y 474.619,Z 346.171,A -85,B 0,C 180,E1 -7140.942,E2 -7140.942} C_VEL
LIN {X 0,Y 474.602,Z 345.989,A -85,B 0,C 180,E1 -7143.977,E2 -7143.977} C_VEL
LIN {X 0,Y 474.547,Z 345.996,A -85,B 0,C 180,E1 -7146.895,E2 -7146.895} C_VEL
LIN {X 0,Y 474.578,Z 345.986,A -85,B 0,C 180,E1 -7149.64,E2 -7149.64} C_VEL
LIN {X 0,Y 474.567,Z 345.992,A -85,B 0,C 180,E1 -7152.94,E2 -7152.94} C_VEL
LIN {X 0,Y 474.601,Z 345.995,A -85,B 0,C 180,E1 -7155.894,E2 -7155.894} C_VEL
LIN {X 0,Y 474.59,Z 345.994,A -85,B 0,C 180,E1 -7159.339,E2 -7159.339} C_VEL
LIN {X 0,Y 474.591,Z 345.992,A -85,B 0,C 180,E1 -7161.707,E2 -7161.707} C_VEL
LIN {X 0,Y 474.616,Z 345.982,A -85,B 0,C 180,E1 -7164.725,E2 -7164.725} C_VEL
LIN {X 0,Y 474.628,Z 345.985,A -85,B 0,C 180,E1 -7167.787,E2 -7167.787} C_VEL
LIN {X 0,Y 474.606,Z 345.988,A -85,B 0,C 180,E1 -7170.889,E2 -7170.889} C_VEL
LIN {X 0,Y 474.59,Z 345.988,A -85,B 0,C 180,E1 -7173.624,E2 -7173.624} C_VEL
LIN {X 0,Y 474.634,Z 345.981,A -85,B 0,C 180,E1 -7176.642,E2 -7176.642} C_VEL
LIN {X 0,Y 474.654,Z 345.984,A -85,B 0,C 180,E1 -7180.089,E2 -7180.089} C_VEL
LIN {X 0,Y 474.635,Z 345.978,A -85,B 0,C 180,E1 -7182.774,E2 -7182.774} C_VEL
LIN {X 0,Y 474.648,Z 345.986,A -85,B 0,C 180,E1 -7185.421,E2 -7185.421} C_VEL
LIN {X 0,Y 474.705,Z 345.969,A -85,B 0,C 180,E1 -7188.038,E2 -7188.038} C_VEL
LIN {X 0,Y 474.712,Z 345.979,A -85,B 0,C 180,E1 -7191.486,E2 -7191.486} C_VEL
LIN {X 0,Y 474.777,Z 345.96,A -85,B 0,C 180,E1 -7194.052,E2 -7194.052} C_VEL
LIN {X 0,Y 474.884,Z 345.957,A -85,B 0,C 180,E1 -7197.455,E2 -7197.455} C_VEL
LIN {X 0,Y 474.912,Z 345.945,A -85,B 0,C 180,E1 -7200,E2 -7200} C_VEL
LIN {X 0,Y 474.888,Z 345.946,A -85,B 0,C 180,E1 -7202.545,E2 -7202.545} C_VEL
LIN {X 0,Y 474.761,Z 345.965,A -85,B 0,C 180,E1 -7205.948,E2 -7205.948} C_VEL
LIN {X 0,Y 474.713,Z 345.965,A -85,B 0,C 180,E1 -7208.514,E2 -7208.514} C_VEL
LIN {X 0,Y 474.705,Z 345.972,A -85,B 0,C 180,E1 -7211.962,E2 -7211.962} C_VEL
LIN {X 0,Y 474.7,Z 345.979,A -85,B 0,C 180,E1 -7215.456,E2 -7215.456} C_VEL
LIN {X 0,Y 474.663,Z 345.979,A -85,B 0,C 180,E1 -7219.01,E2 -7219.01} C_VEL
LIN {X 0,Y 474.589,Z 345.992,A -85,B 0,C 180,E1 -7221.729,E2 -7221.729} C_VEL
LIN {X 0,Y 474.653,Z 345.978,A -85,B 0,C 180,E1 -7224.493,E2 -7224.493} C_VEL
LIN {X 0,Y 474.681,Z 345.984,A -85,B 0,C 180,E1 -7227.334,E2 -7227.334} C_VEL
LIN {X 0,Y 474.605,Z 345.981,A -85,B 0,C 180,E1 -7230.23,E2 -7230.23} C_VEL
LIN {X 0,Y 474.643,Z 345.985,A -85,B 0,C 180,E1 -7233.22,E2 -7233.22} C_VEL
LIN {X 0,Y 474.589,Z 345.99,A -85,B 0,C 180,E1 -7236.323,E2 -7236.323} C_VEL
LIN {X 0,Y 474.618,Z 345.965,A -85,B 0,C 180,E1 -7239.646,E2 -7239.646} C_VEL
LIN {X 0,Y 474.632,Z 345.987,A -85,B 0,C 180,E1 -7242.932,E2 -7242.932} C_VEL
LIN {X 0,Y 474.608,Z 345.977,A -85,B 0,C 180,E1 -7245.895,E2 -7245.895} C_VEL
LIN {X 0,Y 474.628,Z 345.99,A -85,B 0,C 180,E1 -7249.041,E2 -7249.041} C_VEL
LIN {X 0,Y 474.61,Z 345.989,A -85,B 0,C 180,E1 -7251.704,E2 -7251.704} C_VEL
LIN {X 0,Y 474.624,Z 345.992,A -85,B 0,C 180,E1 -7254.726,E2 -7254.726} C_VEL
LIN {X 0,Y 474.635,Z 345.986,A -85,B 0,C 180,E1 -7257.788,E2 -7257.788} C_VEL
LIN {X 0,Y 474.646,Z 346.182,A -85,B 0,C 180,E1 -7259.356,E2 -7259.356} C_VEL
LIN {X 0,Y 478.797,Z 361.576,A -85,B 0,C 180,E1 -7261.728,E2 -7261.728} C_VEL
LIN {X 0,Y 480.195,Z 367.127,A -85,B 0,C 180,E1 -7262.547,E2 -7262.547} C_VEL
LIN {X 0,Y 479.901,Z 375.309,A -85,B 0,C 180,E1 -7263.607,E2 -7263.607} C_VEL
LIN {X 0,Y 478.609,Z 397.574,A -85,B 0,C 180,E1 -7266.413,E2 -7266.413} C_VEL
LIN {X 0,Y 478.81,Z 399.572,A -85,B 0,C 180,E1 -7266.524,E2 -7266.524} C_VEL
LIN {X 0,Y 481.846,Z 417.526,A -85,B 0,C 180,E1 -7266.978,E2 -7266.978} C_VEL
LIN {X 0,Y 480.944,Z 490.026,A -85,B 0,C 180,E1 -7268.122,E2 -7268.122} C_VEL
LIN {X 0,Y 480.179,Z 565.47,A -85,B 0,C 180,E1 -7269.295,E2 -7269.295} C_VEL
LIN {X 0,Y 479.755,Z 580.98,A -85,B 0,C 180,E1 -7269.71,E2 -7269.71} C_VEL
LIN {X 0,Y 479.292,Z 594.519,A -85,B 0,C 180,E1 -7270.23,E2 -7270.23} C_VEL
LIN {X 0,Y 478.584,Z 608.544,A -85,B 0,C 180,E1 -7270.929,E2 -7270.929} C_VEL
LIN {X 0,Y 477.864,Z 622.138,A -85,B 0,C 180,E1 -7271.789,E2 -7271.789} C_VEL
LIN {X 0,Y 477.153,Z 634.618,A -85,B 0,C 180,E1 -7272.757,E2 -7272.757} C_VEL
LIN {X 0,Y 476.481,Z 646.178,A -85,B 0,C 180,E1 -7273.835,E2 -7273.835} C_VEL
LIN {X 0,Y 475.794,Z 656.9,A -85,B 0,C 180,E1 -7275.019,E2 -7275.019} C_VEL
LIN {X 0,Y 475.242,Z 666.797,A -85,B 0,C 180,E1 -7276.313,E2 -7276.313} C_VEL
LIN {X 0,Y 474.695,Z 675.929,A -85,B 0,C 180,E1 -7277.728,E2 -7277.728} C_VEL
LIN {X 0,Y 474.382,Z 684.482,A -85,B 0,C 180,E1 -7279.328,E2 -7279.328} C_VEL
LIN {X 0,Y 474.052,Z 691.955,A -85,B 0,C 180,E1 -7281.045,E2 -7281.045} C_VEL
LIN {X 0,Y 473.9,Z 697.88,A -85,B 0,C 180,E1 -7282.758,E2 -7282.758} C_VEL
LIN {X 0,Y 473.8,Z 701.376,A -85,B 0,C 180,E1 -7284.04,E2 -7284.04} C_VEL
LIN {X 0,Y 473.702,Z 704.925,A -85,B 0,C 180,E1 -7285.746,E2 -7285.746} C_VEL
LIN {X 0,Y 473.755,Z 707.258,A -85,B 0,C 180,E1 -7287.449,E2 -7287.449} C_VEL
LIN {X 0,Y 473.685,Z 708.432,A -85,B 0,C 180,E1 -7289.15,E2 -7289.15} C_VEL
LIN {X 0,Y 473.685,Z 708.432,A -85,B 0,C 180,E1 -7290.85,E2 -7290.85} C_VEL
LIN {X 0,Y 473.765,Z 707.26,A -85,B 0,C 180,E1 -7292.551,E2 -7292.551} C_VEL
LIN {X 0,Y 473.704,Z 704.925,A -85,B 0,C 180,E1 -7294.254,E2 -7294.254} C_VEL
LIN {X 0,Y 473.787,Z 701.372,A -85,B 0,C 180,E1 -7295.96,E2 -7295.96} C_VEL
LIN {X 0,Y 473.933,Z 696.517,A -85,B 0,C 180,E1 -7297.67,E2 -7297.67} C_VEL
LIN {X 0,Y 474.124,Z 690.233,A -85,B 0,C 180,E1 -7299.384,E2 -7299.384} C_VEL
LIN {X 0,Y 474.472,Z 682.326,A -85,B 0,C 180,E1 -7301.102,E2 -7301.102} C_VEL
LIN {X 0,Y 474.88,Z 673.673,A -85,B 0,C 180,E1 -7302.641,E2 -7302.641} C_VEL
LIN {X 0,Y 475.431,Z 663.674,A -85,B 0,C 180,E1 -7304.118,E2 -7304.118} C_VEL
LIN {X 0,Y 475.995,Z 653.215,A -85,B 0,C 180,E1 -7305.413,E2 -7305.413} C_VEL
LIN {X 0,Y 476.807,Z 641.222,A -85,B 0,C 180,E1 -7306.649,E2 -7306.649} C_VEL
LIN {X 0,Y 477.474,Z 629.375,A -85,B 0,C 180,E1 -7307.673,E2 -7307.673} C_VEL
LIN {X 0,Y 478.202,Z 617.405,A -85,B 0,C 180,E1 -7308.531,E2 -7308.531} C_VEL
LIN {X 0,Y 478.858,Z 603.588,A -85,B 0,C 180,E1 -7309.338,E2 -7309.338} C_VEL
LIN {X 0,Y 479.48,Z 588.624,A -85,B 0,C 180,E1 -7310.016,E2 -7310.016} C_VEL
LIN {X 0,Y 479.979,Z 573.179,A -85,B 0,C 180,E1 -7310.521,E2 -7310.521} C_VEL
LIN {X 0,Y 480.307,Z 558.025,A -85,B 0,C 180,E1 -7310.839,E2 -7310.839} C_VEL
LIN {X 0,Y 481.782,Z 417.653,A -85,B 0,C 180,E1 -7312.999,E2 -7312.999} C_VEL
LIN {X 0,Y 478.703,Z 398.369,A -85,B 0,C 180,E1 -7313.554,E2 -7313.554} C_VEL
LIN {X 0,Y 480.093,Z 377.836,A -85,B 0,C 180,E1 -7316.227,E2 -7316.227} C_VEL
LIN {X 0,Y 480.825,Z 369.078,A -85,B 0,C 180,E1 -7317.414,E2 -7317.414} C_VEL
LIN {X 0,Y 478.308,Z 358.329,A -85,B 0,C 180,E1 -7319.209,E2 -7319.209} C_VEL
LIN {X 0,Y 475.085,Z 347.823,A -85,B 0,C 180,E1 -7321.182,E2 -7321.182} C_VEL
LIN {X 0,Y 474.609,Z 346.072,A -85,B 0,C 180,E1 -7321.59,E2 -7321.59} C_VEL
LIN {X 0,Y 474.634,Z 345.988,A -85,B 0,C 180,E1 -7324.241,E2 -7324.241} C_VEL
LIN {X 0,Y 474.591,Z 345.995,A -85,B 0,C 180,E1 -7327.384,E2 -7327.384} C_VEL
LIN {X 0,Y 474.628,Z 345.989,A -85,B 0,C 180,E1 -7329.648,E2 -7329.648} C_VEL
LIN {X 0,Y 474.607,Z 345.994,A -85,B 0,C 180,E1 -7332.935,E2 -7332.935} C_VEL
LIN {X 0,Y 474.604,Z 345.992,A -85,B 0,C 180,E1 -7335.895,E2 -7335.895} C_VEL
LIN {X 0,Y 474.623,Z 345.99,A -85,B 0,C 180,E1 -7339.042,E2 -7339.042} C_VEL
LIN {X 0,Y 474.608,Z 345.992,A -85,B 0,C 180,E1 -7341.705,E2 -7341.705} C_VEL
LIN {X 0,Y 474.621,Z 345.992,A -85,B 0,C 180,E1 -7344.725,E2 -7344.725} C_VEL
LIN {X 0,Y 474.636,Z 345.989,A -85,B 0,C 180,E1 -7347.788,E2 -7347.788} C_VEL
LIN {X 0,Y 474.632,Z 346.174,A -85,B 0,C 180,E1 -7350.063,E2 -7350.063} C_VEL
LIN {X 0,Y 477.564,Z 356.698,A -85,B 0,C 180,E1 -7352.328,E2 -7352.328} C_VEL
LIN {X 0,Y 479.616,Z 366.074,A -85,B 0,C 180,E1 -7354.155,E2 -7354.155} C_VEL
LIN {X 0,Y 479.393,Z 371.322,A -85,B 0,C 180,E1 -7355.039,E2 -7355.039} C_VEL
LIN {X 0,Y 478.018,Z 391.064,A -85,B 0,C 180,E1 -7358.215,E2 -7358.215} C_VEL
LIN {X 0,Y 477.649,Z 398.138,A -85,B 0,C 180,E1 -7359.293,E2 -7359.293} C_VEL
LIN {X 0,Y 480.675,Z 413.363,A -85,B 0,C 180,E1 -7359.806,E2 -7359.806} C_VEL
LIN {X 0,Y 481.125,Z 417.993,A -85,B 0,C 180,E1 -7359.926,E2 -7359.926} C_VEL
LIN {X 0,Y 479.214,Z 511.679,A -85,B 0,C 180,E1 -7361.676,E2 -7361.676} C_VEL
LIN {X 0,Y 478.676,Z 540.685,A -85,B 0,C 180,E1 -7362.224,E2 -7362.224} C_VEL
LIN {X 0,Y 478.258,Z 555.649,A -85,B 0,C 180,E1 -7362.686,E2 -7362.686} C_VEL
LIN {X 0,Y 477.857,Z 569.027,A -85,B 0,C 180,E1 -7363.268,E2 -7363.268} C_VEL
LIN {X 0,Y 477.358,Z 581.61,A -85,B 0,C 180,E1 -7363.975,E2 -7363.975} C_VEL
LIN {X 0,Y 476.793,Z 593.88,A -85,B 0,C 180,E1 -7364.833,E2 -7364.833} C_VEL
LIN {X 0,Y 476.261,Z 605.163,A -85,B 0,C 180,E1 -7365.799,E2 -7365.799} C_VEL
LIN {X 0,Y 475.676,Z 616.504,A -85,B 0,C 180,E1 -7366.979,E2 -7366.979} C_VEL
LIN {X 0,Y 475.205,Z 626.638,A -85,B 0,C 180,E1 -7368.267,E2 -7368.267} C_VEL
LIN {X 0,Y 474.744,Z 635.042,A -85,B 0,C 180,E1 -7369.552,E2 -7369.552} C_VEL
LIN {X 0,Y 474.419,Z 643.044,A -85,B 0,C 180,E1 -7371.052,E2 -7371.052} C_VEL
LIN {X 0,Y 474.165,Z 648.647,A -85,B 0,C 180,E1 -7372.334,E2 -7372.334} C_VEL
LIN {X 0,Y 474.053,Z 654.487,A -85,B 0,C 180,E1 -7374.043,E2 -7374.043} C_VEL
LIN {X 0,Y 473.848,Z 656.803,A -85,B 0,C 180,E1 -7374.895,E2 -7374.895} C_VEL
LIN {X 0,Y 473.902,Z 658.724,A -85,B 0,C 180,E1 -7375.748,E2 -7375.748} C_VEL
LIN {X 0,Y 473.833,Z 661.486,A -85,B 0,C 180,E1 -7377.45,E2 -7377.45} C_VEL
LIN {X 0,Y 473.686,Z 662.858,A -85,B 0,C 180,E1 -7379.15,E2 -7379.15} C_VEL
LIN {X 0,Y 473.686,Z 662.855,A -85,B 0,C 180,E1 -7380.85,E2 -7380.85} C_VEL
LIN {X 0,Y 473.806,Z 661.474,A -85,B 0,C 180,E1 -7382.551,E2 -7382.551} C_VEL
LIN {X 0,Y 473.869,Z 658.698,A -85,B 0,C 180,E1 -7384.253,E2 -7384.253} C_VEL
LIN {X 0,Y 474.036,Z 654.452,A -85,B 0,C 180,E1 -7385.957,E2 -7385.957} C_VEL
LIN {X 0,Y 474.132,Z 648.628,A -85,B 0,C 180,E1 -7387.667,E2 -7387.667} C_VEL
LIN {X 0,Y 474.406,Z 642.048,A -85,B 0,C 180,E1 -7389.164,E2 -7389.164} C_VEL
LIN {X 0,Y 474.745,Z 633.866,A -85,B 0,C 180,E1 -7390.664,E2 -7390.664} C_VEL
LIN {X 0,Y 475.282,Z 624.212,A -85,B 0,C 180,E1 -7392.095,E2 -7392.095} C_VEL
LIN {X 0,Y 475.66,Z 614.93,A -85,B 0,C 180,E1 -7393.239,E2 -7393.239} C_VEL
LIN {X 0,Y 476.284,Z 603.315,A -85,B 0,C 180,E1 -7394.419,E2 -7394.419} C_VEL
LIN {X 0,Y 476.838,Z 591.764,A -85,B 0,C 180,E1 -7395.385,E2 -7395.385} C_VEL
LIN {X 0,Y 477.397,Z 579.142,A -85,B 0,C 180,E1 -7396.243,E2 -7396.243} C_VEL
LIN {X 0,Y 477.949,Z 566.114,A -85,B 0,C 180,E1 -7396.943,E2 -7396.943} C_VEL
LIN {X 0,Y 478.368,Z 552.126,A -85,B 0,C 180,E1 -7397.515,E2 -7397.515} C_VEL
LIN {X 0,Y 478.728,Z 537.017,A -85,B 0,C 180,E1 -7397.941,E2 -7397.941} C_VEL
LIN {X 0,Y 480.407,Z 416.103,A -85,B 0,C 180,E1 -7399.991,E2 -7399.991} C_VEL
LIN {X 0,Y 477.123,Z 397.781,A -85,B 0,C 180,E1 -7400.481,E2 -7400.481} C_VEL
LIN {X 0,Y 477.709,Z 384.372,A -85,B 0,C 180,E1 -7402.489,E2 -7402.489} C_VEL
LIN {X 0,Y 478.725,Z 365.306,A -85,B 0,C 180,E1 -7405.43,E2 -7405.43} C_VEL
LIN {X 0,Y 478.006,Z 360.397,A -85,B 0,C 180,E1 -7406.25,E2 -7406.25} C_VEL
LIN {X 0,Y 474.633,Z 346.261,A -85,B 0,C 180,E1 -7408.766,E2 -7408.766} C_VEL
LIN {X 0,Y 474.572,Z 345.995,A -85,B 0,C 180,E1 -7409.255,E2 -7409.255} C_VEL
LIN {X 0,Y 474.584,Z 345.997,A -85,B 0,C 180,E1 -7412.424,E2 -7412.424} C_VEL
LIN {X 0,Y 474.592,Z 345.992,A -85,B 0,C 180,E1 -7415.465,E2 -7415.465} C_VEL
LIN {X 0,Y 474.584,Z 345.994,A -85,B 0,C 180,E1 -7418.46,E2 -7418.46} C_VEL
LIN {X 0,Y 474.581,Z 345.99,A -85,B 0,C 180,E1 -7421.79,E2 -7421.79} C_VEL
LIN {X 0,Y 474.613,Z 345.989,A -85,B 0,C 180,E1 -7425.298,E2 -7425.298} C_VEL
LIN {X 0,Y 474.58,Z 345.995,A -85,B 0,C 180,E1 -7428.21,E2 -7428.21} C_VEL
LIN {X 0,Y 474.572,Z 345.989,A -85,B 0,C 180,E1 -7430.887,E2 -7430.887} C_VEL
LIN {X 0,Y 473.9,Z 346.078,A -85,B 0,C 180,E1 -7431.595,E2 -7431.595} C_VEL
LIN {X 0,Y 471.052,Z 346.434,A -85,B 0,C 180,E1 -7432.744,E2 -7432.744} C_VEL
LIN {X 0,Y 468.647,Z 346.735,A -85,B 0,C 180,E1 -7433.671,E2 -7433.671} C_VEL
LIN {X 0,Y 467.614,Z 346.865,A -85,B 0,C 180,E1 -7434.387,E2 -7434.387} C_VEL
LIN {X 0,Y 467.529,Z 346.872,A -85,B 0,C 180,E1 -7434.63,E2 -7434.63} C_VEL
LIN {X 0,Y 467.547,Z 346.87,A -85,B 0,C 180,E1 -7437.328,E2 -7437.328} C_VEL
LIN {X 0,Y 467.563,Z 347.062,A -85,B 0,C 180,E1 -7438.827,E2 -7438.827} C_VEL
LIN {X 0,Y 471.559,Z 362.651,A -85,B 0,C 180,E1 -7441.273,E2 -7441.273} C_VEL
LIN {X 0,Y 472.699,Z 367.954,A -85,B 0,C 180,E1 -7442.074,E2 -7442.074} C_VEL
LIN {X 0,Y 471.972,Z 387.333,A -85,B 0,C 180,E1 -7444.652,E2 -7444.652} C_VEL
LIN {X 0,Y 471.609,Z 397.752,A -85,B 0,C 180,E1 -7445.938,E2 -7445.938} C_VEL
LIN {X 0,Y 475.887,Z 419.911,A -85,B 0,C 180,E1 -7446.533,E2 -7446.533} C_VEL
LIN {X 0,Y 474.252,Z 564.439,A -85,B 0,C 180,E1 -7448.796,E2 -7448.796} C_VEL
LIN {X 0,Y 473.751,Z 579.965,A -85,B 0,C 180,E1 -7449.2,E2 -7449.2} C_VEL
LIN {X 0,Y 473.139,Z 594.702,A -85,B 0,C 180,E1 -7449.759,E2 -7449.759} C_VEL
LIN {X 0,Y 472.435,Z 608.422,A -85,B 0,C 180,E1 -7450.445,E2 -7450.445} C_VEL
LIN {X 0,Y 471.664,Z 622.182,A -85,B 0,C 180,E1 -7451.315,E2 -7451.315} C_VEL
LIN {X 0,Y 470.792,Z 634.81,A -85,B 0,C 180,E1 -7452.292,E2 -7452.292} C_VEL
LIN {X 0,Y 469.989,Z 647.569,A -85,B 0,C 180,E1 -7453.494,E2 -7453.494} C_VEL
LIN {X 0,Y 469.137,Z 659.145,A -85,B 0,C 180,E1 -7454.801,E2 -7454.801} C_VEL
LIN {X 0,Y 468.478,Z 668.896,A -85,B 0,C 180,E1 -7456.112,E2 -7456.112} C_VEL
LIN {X 0,Y 467.848,Z 678.763,A -85,B 0,C 180,E1 -7457.698,E2 -7457.698} C_VEL
LIN {X 0,Y 467.493,Z 686.392,A -85,B 0,C 180,E1 -7459.169,E2 -7459.169} C_VEL
LIN {X 0,Y 467.065,Z 693.8,A -85,B 0,C 180,E1 -7460.909,E2 -7460.909} C_VEL
LIN {X 0,Y 466.828,Z 699.682,A -85,B 0,C 180,E1 -7462.648,E2 -7462.648} C_VEL
LIN {X 0,Y 466.73,Z 703.158,A -85,B 0,C 180,E1 -7463.949,E2 -7463.949} C_VEL
LIN {X 0,Y 466.618,Z 706.706,A -85,B 0,C 180,E1 -7465.681,E2 -7465.681} C_VEL
LIN {X 0,Y 466.639,Z 709.049,A -85,B 0,C 180,E1 -7467.41,E2 -7467.41} C_VEL
LIN {X 0,Y 466.586,Z 710.241,A -85,B 0,C 180,E1 -7469.137,E2 -7469.137} C_VEL
LIN {X 0,Y 466.587,Z 710.257,A -85,B 0,C 180,E1 -7470.863,E2 -7470.863} C_VEL
LIN {X 0,Y 466.64,Z 709.127,A -85,B 0,C 180,E1 -7472.59,E2 -7472.59} C_VEL
LIN {X 0,Y 466.618,Z 706.851,A -85,B 0,C 180,E1 -7474.319,E2 -7474.319} C_VEL
LIN {X 0,Y 466.752,Z 703.378,A -85,B 0,C 180,E1 -7476.05,E2 -7476.05} C_VEL
LIN {X 0,Y 466.885,Z 698.62,A -85,B 0,C 180,E1 -7477.786,E2 -7477.786} C_VEL
LIN {X 0,Y 467.121,Z 692.449,A -85,B 0,C 180,E1 -7479.526,E2 -7479.526} C_VEL
LIN {X 0,Y 467.605,Z 684.694,A -85,B 0,C 180,E1 -7481.267,E2 -7481.267} C_VEL
LIN {X 0,Y 468.001,Z 676.312,A -85,B 0,C 180,E1 -7482.817,E2 -7482.817} C_VEL
LIN {X 0,Y 468.665,Z 666.474,A -85,B 0,C 180,E1 -7484.325,E2 -7484.325} C_VEL
LIN {X 0,Y 469.306,Z 656.313,A -85,B 0,C 180,E1 -7485.638,E2 -7485.638} C_VEL
LIN {X 0,Y 470.141,Z 644.453,A -85,B 0,C 180,E1 -7486.918,E2 -7486.918} C_VEL
LIN {X 0,Y 470.999,Z 632.006,A -85,B 0,C 180,E1 -7488.036,E2 -7488.036} C_VEL
LIN {X 0,Y 471.872,Z 618.765,A -85,B 0,C 180,E1 -7489.014,E2 -7489.014} C_VEL
LIN {X 0,Y 472.645,Z 605.16,A -85,B 0,C 180,E1 -7489.829,E2 -7489.829} C_VEL
LIN {X 0,Y 473.35,Z 589.678,A -85,B 0,C 180,E1 -7490.548,E2 -7490.548} C_VEL
LIN {X 0,Y 473.932,Z 574.898,A -85,B 0,C 180,E1 -7491.047,E2 -7491.047} C_VEL
LIN {X 0,Y 474.315,Z 559.075,A -85,B 0,C 180,E1 -7491.4,E2 -7491.4} C_VEL
LIN {X 0,Y 475.91,Z 420.061,A -85,B 0,C 180,E1 -7493.555,E2 -7493.555} C_VEL
LIN {X 0,Y 471.612,Z 397.434,A -85,B 0,C 180,E1 -7494.172,E2 -7494.172} C_VEL
LIN {X 0,Y 472.259,Z 379.198,A -85,B 0,C 180,E1 -7496.516,E2 -7496.516} C_VEL
LIN {X 0,Y 472.717,Z 368.653,A -85,B 0,C 180,E1 -7497.925,E2 -7497.925} C_VEL
LIN {X 0,Y 470.361,Z 357.97,A -85,B 0,C 180,E1 -7499.543,E2 -7499.543} C_VEL
LIN {X 0,Y 467.565,Z 346.983,A -85,B 0,C 180,E1 -7501.3,E2 -7501.3} C_VEL
LIN {X 0,Y 467.561,Z 346.869,A -85,B 0,C 180,E1 -7504.237,E2 -7504.237} C_VEL
LIN {X 0,Y 467.512,Z 346.873,A -85,B 0,C 180,E1 -7507.18,E2 -7507.18} C_VEL
LIN {X 0,Y 467.516,Z 346.869,A -85,B 0,C 180,E1 -7510.271,E2 -7510.271} C_VEL
LIN {X 0,Y 467.516,Z 346.871,A -85,B 0,C 180,E1 -7512.568,E2 -7512.568} C_VEL
LIN {X 0,Y 467.565,Z 346.864,A -85,B 0,C 180,E1 -7515.052,E2 -7515.052} C_VEL
LIN {X 0,Y 467.559,Z 346.867,A -85,B 0,C 180,E1 -7518.726,E2 -7518.726} C_VEL
LIN {X 0,Y 467.542,Z 346.874,A -85,B 0,C 180,E1 -7521.953,E2 -7521.953} C_VEL
LIN {X 0,Y 467.553,Z 346.863,A -85,B 0,C 180,E1 -7525.166,E2 -7525.166} C_VEL
LIN {X 0,Y 467.579,Z 346.859,A -85,B 0,C 180,E1 -7528.259,E2 -7528.259} C_VEL
LIN {X 0,Y 467.554,Z 346.869,A -85,B 0,C 180,E1 -7531.249,E2 -7531.249} C_VEL
LIN {X 0,Y 467.567,Z 346.866,A -85,B 0,C 180,E1 -7534.157,E2 -7534.157} C_VEL
LIN {X 0,Y 467.576,Z 346.862,A -85,B 0,C 180,E1 -7536.996,E2 -7536.996} C_VEL
LIN {X 0,Y 467.622,Z 346.863,A -85,B 0,C 180,E1 -7539.777,E2 -7539.777} C_VEL
LIN {X 0,Y 467.595,Z 346.854,A -85,B 0,C 180,E1 -7542.506,E2 -7542.506} C_VEL
LIN {X 0,Y 467.606,Z 346.86,A -85,B 0,C 180,E1 -7545.196,E2 -7545.196} C_VEL
LIN {X 0,Y 467.657,Z 346.849,A -85,B 0,C 180,E1 -7547.854,E2 -7547.854} C_VEL
LIN {X 0,Y 467.67,Z 346.854,A -85,B 0,C 180,E1 -7551.357,E2 -7551.357} C_VEL
LIN {X 0,Y 467.741,Z 346.837,A -85,B 0,C 180,E1 -7553.962,E2 -7553.962} C_VEL
LIN {X 0,Y 467.849,Z 346.833,A -85,B 0,C 180,E1 -7557.417,E2 -7557.417} C_VEL
LIN {X 0,Y 467.882,Z 346.821,A -85,B 0,C 180,E1 -7560,E2 -7560} C_VEL
LIN {X 0,Y 467.853,Z 346.822,A -85,B 0,C 180,E1 -7562.583,E2 -7562.583} C_VEL
LIN {X 0,Y 467.724,Z 346.841,A -85,B 0,C 180,E1 -7566.038,E2 -7566.038} C_VEL
LIN {X 0,Y 467.662,Z 346.855,A -85,B 0,C 180,E1 -7569.515,E2 -7569.515} C_VEL
LIN {X 0,Y 467.655,Z 346.849,A -85,B 0,C 180,E1 -7572.357,E2 -7572.357} C_VEL
LIN {X 0,Y 467.65,Z 346.854,A -85,B 0,C 180,E1 -7575.885,E2 -7575.885} C_VEL
LIN {X 0,Y 467.623,Z 346.853,A -85,B 0,C 180,E1 -7579.308,E2 -7579.308} C_VEL
LIN {X 0,Y 467.535,Z 346.869,A -85,B 0,C 180,E1 -7582.074,E2 -7582.074} C_VEL
LIN {X 0,Y 467.593,Z 346.858,A -85,B 0,C 180,E1 -7584.888,E2 -7584.888} C_VEL
LIN {X 0,Y 467.62,Z 346.859,A -85,B 0,C 180,E1 -7587.769,E2 -7587.769} C_VEL
LIN {X 0,Y 467.568,Z 346.865,A -85,B 0,C 180,E1 -7591.045,E2 -7591.045} C_VEL
LIN {X 0,Y 467.588,Z 346.857,A -85,B 0,C 180,E1 -7594.242,E2 -7594.242} C_VEL
LIN {X 0,Y 467.548,Z 346.869,A -85,B 0,C 180,E1 -7597.186,E2 -7597.186} C_VEL
LIN {X 0,Y 467.575,Z 346.84,A -85,B 0,C 180,E1 -7600.265,E2 -7600.265} C_VEL
LIN {X 0,Y 467.586,Z 346.859,A -85,B 0,C 180,E1 -7602.567,E2 -7602.567} C_VEL
LIN {X 0,Y 467.57,Z 346.861,A -85,B 0,C 180,E1 -7605.053,E2 -7605.053} C_VEL
LIN {X 0,Y 467.589,Z 346.852,A -85,B 0,C 180,E1 -7607.44,E2 -7607.44} C_VEL
LIN {X 0,Y 467.583,Z 346.869,A -85,B 0,C 180,E1 -7610.855,E2 -7610.855} C_VEL
LIN {X 0,Y 467.559,Z 346.868,A -85,B 0,C 180,E1 -7614.261,E2 -7614.261} C_VEL
LIN {X 0,Y 467.582,Z 346.868,A -85,B 0,C 180,E1 -7617.321,E2 -7617.321} C_VEL
LIN {X 0,Y 467.584,Z 347.093,A -85,B 0,C 180,E1 -7619.016,E2 -7619.016} C_VEL
LIN {X 0,Y 471.982,Z 363.244,A -85,B 0,C 180,E1 -7621.543,E2 -7621.543} C_VEL
LIN {X 0,Y 473.361,Z 368.675,A -85,B 0,C 180,E1 -7622.357,E2 -7622.357} C_VEL
LIN {X 0,Y 473.373,Z 373.283,A -85,B 0,C 180,E1 -7622.974,E2 -7622.974} C_VEL
LIN {X 0,Y 471.828,Z 397.798,A -85,B 0,C 180,E1 -7626.111,E2 -7626.111} C_VEL
LIN {X 0,Y 472.482,Z 402.026,A -85,B 0,C 180,E1 -7626.261,E2 -7626.261} C_VEL
LIN {X 0,Y 475.242,Z 418.556,A -85,B 0,C 180,E1 -7626.687,E2 -7626.687} C_VEL
LIN {X 0,Y 473.556,Z 565.592,A -85,B 0,C 180,E1 -7628.992,E2 -7628.992} C_VEL
LIN {X 0,Y 473.113,Z 580.936,A -85,B 0,C 180,E1 -7629.408,E2 -7629.408} C_VEL
LIN {X 0,Y 472.628,Z 593.327,A -85,B 0,C 180,E1 -7629.884,E2 -7629.884} C_VEL
LIN {X 0,Y 471.979,Z 606.616,A -85,B 0,C 180,E1 -7630.539,E2 -7630.539} C_VEL
LIN {X 0,Y 471.229,Z 620.601,A -85,B 0,C 180,E1 -7631.41,E2 -7631.41} C_VEL
LIN {X 0,Y 470.409,Z 633.364,A -85,B 0,C 180,E1 -7632.39,E2 -7632.39} C_VEL
LIN {X 0,Y 469.597,Z 646.207,A -85,B 0,C 180,E1 -7633.592,E2 -7633.592} C_VEL
LIN {X 0,Y 468.892,Z 656.925,A -85,B 0,C 180,E1 -7634.794,E2 -7634.794} C_VEL
LIN {X 0,Y 468.3,Z 666.821,A -85,B 0,C 180,E1 -7636.106,E2 -7636.106} C_VEL
LIN {X 0,Y 467.669,Z 676.472,A -85,B 0,C 180,E1 -7637.634,E2 -7637.634} C_VEL
LIN {X 0,Y 467.366,Z 684.501,A -85,B 0,C 180,E1 -7639.166,E2 -7639.166} C_VEL
LIN {X 0,Y 467.012,Z 691.973,A -85,B 0,C 180,E1 -7640.909,E2 -7640.909} C_VEL
LIN {X 0,Y 466.817,Z 697.896,A -85,B 0,C 180,E1 -7642.648,E2 -7642.648} C_VEL
LIN {X 0,Y 466.715,Z 701.389,A -85,B 0,C 180,E1 -7643.949,E2 -7643.949} C_VEL
LIN {X 0,Y 466.615,Z 704.936,A -85,B 0,C 180,E1 -7645.681,E2 -7645.681} C_VEL
LIN {X 0,Y 466.673,Z 707.27,A -85,B 0,C 180,E1 -7647.411,E2 -7647.411} C_VEL
LIN {X 0,Y 466.587,Z 708.446,A -85,B 0,C 180,E1 -7649.137,E2 -7649.137} C_VEL
LIN {X 0,Y 466.587,Z 708.446,A -85,B 0,C 180,E1 -7650.863,E2 -7650.863} C_VEL
LIN {X 0,Y 466.681,Z 707.274,A -85,B 0,C 180,E1 -7652.59,E2 -7652.59} C_VEL
LIN {X 0,Y 466.617,Z 704.94,A -85,B 0,C 180,E1 -7654.319,E2 -7654.319} C_VEL
LIN {X 0,Y 466.703,Z 701.387,A -85,B 0,C 180,E1 -7656.051,E2 -7656.051} C_VEL
LIN {X 0,Y 466.868,Z 696.533,A -85,B 0,C 180,E1 -7657.787,E2 -7657.787} C_VEL
LIN {X 0,Y 467.065,Z 690.251,A -85,B 0,C 180,E1 -7659.528,E2 -7659.528} C_VEL
LIN {X 0,Y 467.465,Z 682.344,A -85,B 0,C 180,E1 -7661.271,E2 -7661.271} C_VEL
LIN {X 0,Y 467.903,Z 673.821,A -85,B 0,C 180,E1 -7662.812,E2 -7662.812} C_VEL
LIN {X 0,Y 468.478,Z 663.695,A -85,B 0,C 180,E1 -7664.331,E2 -7664.331} C_VEL
LIN {X 0,Y 469.106,Z 653.238,A -85,B 0,C 180,E1 -7665.645,E2 -7665.645} C_VEL
LIN {X 0,Y 469.936,Z 641.902,A -85,B 0,C 180,E1 -7666.837,E2 -7666.837} C_VEL
LIN {X 0,Y 470.666,Z 629.406,A -85,B 0,C 180,E1 -7667.937,E2 -7667.937} C_VEL
LIN {X 0,Y 471.528,Z 615.751,A -85,B 0,C 180,E1 -7668.916,E2 -7668.916} C_VEL
LIN {X 0,Y 472.288,Z 601.501,A -85,B 0,C 180,E1 -7669.731,E2 -7669.731} C_VEL
LIN {X 0,Y 472.897,Z 586.528,A -85,B 0,C 180,E1 -7670.39,E2 -7670.39} C_VEL
LIN {X 0,Y 473.416,Z 571.18,A -85,B 0,C 180,E1 -7670.872,E2 -7670.872} C_VEL
LIN {X 0,Y 473.718,Z 556.409,A -85,B 0,C 180,E1 -7671.172,E2 -7671.172} C_VEL
LIN {X 0,Y 475.225,Z 420.913,A -85,B 0,C 180,E1 -7673.287,E2 -7673.287} C_VEL
LIN {X 0,Y 475.143,Z 417.131,A -85,B 0,C 180,E1 -7673.367,E2 -7673.367} C_VEL
LIN {X 0,Y 472.049,Z 398.418,A -85,B 0,C 180,E1 -7673.936,E2 -7673.936} C_VEL
LIN {X 0,Y 473.53,Z 378.457,A -85,B 0,C 180,E1 -7676.595,E2 -7676.595} C_VEL
LIN {X 0,Y 474.208,Z 371.323,A -85,B 0,C 180,E1 -7677.59,E2 -7677.59} C_VEL
LIN {X 0,Y 471.728,Z 360.508,A -85,B 0,C 180,E1 -7679.449,E2 -7679.449} C_VEL
LIN {X 0,Y 468.831,Z 350.986,A -85,B 0,C 180,E1 -7681.3,E2 -7681.3} C_VEL
LIN {X 0,Y 467.612,Z 346.964,A -85,B 0,C 180,E1 -7682.182,E2 -7682.182} C_VEL
LIN {X 0,Y 467.567,Z 346.871,A -85,B 0,C 180,E1 -7684.833,E2 -7684.833} C_VEL
LIN {X 0,Y 467.566,Z 346.87,A -85,B 0,C 180,E1 -7688.045,E2 -7688.045} C_VEL
LIN {X 0,Y 467.579,Z 346.868,A -85,B 0,C 180,E1 -7691.277,E2 -7691.277} C_VEL
LIN {X 0,Y 467.55,Z 346.87,A -85,B 0,C 180,E1 -7693.82,E2 -7693.82} C_VEL
LIN {X 0,Y 467.549,Z 346.873,A -85,B 0,C 180,E1 -7696.255,E2 -7696.255} C_VEL
LIN {X 0,Y 467.571,Z 346.868,A -85,B 0,C 180,E1 -7699.735,E2 -7699.735} C_VEL
LIN {X 0,Y 467.543,Z 346.874,A -85,B 0,C 180,E1 -7702.815,E2 -7702.815} C_VEL
LIN {X 0,Y 467.582,Z 346.869,A -85,B 0,C 180,E1 -7706.212,E2 -7706.212} C_VEL
LIN {X 0,Y 467.581,Z 346.977,A -85,B 0,C 180,E1 -7709.423,E2 -7709.423} C_VEL
LIN {X 0,Y 470.051,Z 355.617,A -85,B 0,C 180,E1 -7711.416,E2 -7711.416} C_VEL
LIN {X 0,Y 472.532,Z 365.691,A -85,B 0,C 180,E1 -7713.5,E2 -7713.5} C_VEL
LIN {X 0,Y 473.078,Z 369.621,A -85,B 0,C 180,E1 -7714.244,E2 -7714.244} C_VEL
LIN {X 0,Y 471.416,Z 390.832,A -85,B 0,C 180,E1 -7717.737,E2 -7717.737} C_VEL
LIN {X 0,Y 470.974,Z 398.031,A -85,B 0,C 180,E1 -7718.871,E2 -7718.871} C_VEL
LIN {X 0,Y 473.542,Z 410.626,A -85,B 0,C 180,E1 -7719.342,E2 -7719.342} C_VEL
LIN {X 0,Y 474.665,Z 418.106,A -85,B 0,C 180,E1 -7719.57,E2 -7719.57} C_VEL
LIN {X 0,Y 472.589,Z 508.609,A -85,B 0,C 180,E1 -7721.325,E2 -7721.325} C_VEL
LIN {X 0,Y 471.959,Z 541.271,A -85,B 0,C 180,E1 -7721.962,E2 -7721.962} C_VEL
LIN {X 0,Y 471.493,Z 556.034,A -85,B 0,C 180,E1 -7722.429,E2 -7722.429} C_VEL
LIN {X 0,Y 471.047,Z 569.764,A -85,B 0,C 180,E1 -7723.041,E2 -7723.041} C_VEL
LIN {X 0,Y 470.451,Z 583.605,A -85,B 0,C 180,E1 -7723.845,E2 -7723.845} C_VEL
LIN {X 0,Y 469.783,Z 596.821,A -85,B 0,C 180,E1 -7724.823,E2 -7724.823} C_VEL
LIN {X 0,Y 469.173,Z 608.714,A -85,B 0,C 180,E1 -7725.912,E2 -7725.912} C_VEL
LIN {X 0,Y 468.545,Z 619.871,A -85,B 0,C 180,E1 -7727.156,E2 -7727.156} C_VEL
LIN {X 0,Y 468.068,Z 629.937,A -85,B 0,C 180,E1 -7728.525,E2 -7728.525} C_VEL
LIN {X 0,Y 467.652,Z 637.833,A -85,B 0,C 180,E1 -7729.829,E2 -7729.829} C_VEL
LIN {X 0,Y 467.295,Z 645.384,A -85,B 0,C 180,E1 -7731.35,E2 -7731.35} C_VEL
LIN {X 0,Y 467.08,Z 650.605,A -85,B 0,C 180,E1 -7732.652,E2 -7732.652} C_VEL
LIN {X 0,Y 466.908,Z 656.073,A -85,B 0,C 180,E1 -7734.385,E2 -7734.385} C_VEL
LIN {X 0,Y 466.813,Z 659.074,A -85,B 0,C 180,E1 -7735.683,E2 -7735.683} C_VEL
LIN {X 0,Y 466.747,Z 661.837,A -85,B 0,C 180,E1 -7737.411,E2 -7737.411} C_VEL
LIN {X 0,Y 466.617,Z 663.205,A -85,B 0,C 180,E1 -7739.137,E2 -7739.137} C_VEL
LIN {X 0,Y 466.618,Z 663.192,A -85,B 0,C 180,E1 -7740.863,E2 -7740.863} C_VEL
LIN {X 0,Y 466.722,Z 661.793,A -85,B 0,C 180,E1 -7742.589,E2 -7742.589} C_VEL
LIN {X 0,Y 466.778,Z 658.993,A -85,B 0,C 180,E1 -7744.318,E2 -7744.318} C_VEL
LIN {X 0,Y 466.957,Z 654.715,A -85,B 0,C 180,E1 -7746.048,E2 -7746.048} C_VEL
LIN {X 0,Y 467.067,Z 648.851,A -85,B 0,C 180,E1 -7747.783,E2 -7747.783} C_VEL
LIN {X 0,Y 467.374,Z 642.23,A -85,B 0,C 180,E1 -7749.303,E2 -7749.303} C_VEL
LIN {X 0,Y 467.746,Z 634.004,A -85,B 0,C 180,E1 -7750.825,E2 -7750.825} C_VEL
LIN {X 0,Y 468.272,Z 625.382,A -85,B 0,C 180,E1 -7752.129,E2 -7752.129} C_VEL
LIN {X 0,Y 468.712,Z 614.935,A -85,B 0,C 180,E1 -7753.439,E2 -7753.439} C_VEL
LIN {X 0,Y 469.391,Z 603.245,A -85,B 0,C 180,E1 -7754.635,E2 -7754.635} C_VEL
LIN {X 0,Y 469.985,Z 591.61,A -85,B 0,C 180,E1 -7755.615,E2 -7755.615} C_VEL
LIN {X 0,Y 470.549,Z 578.885,A -85,B 0,C 180,E1 -7756.486,E2 -7756.486} C_VEL
LIN {X 0,Y 471.137,Z 565.73,A -85,B 0,C 180,E1 -7757.195,E2 -7757.195} C_VEL
LIN {X 0,Y 471.554,Z 551.94,A -85,B 0,C 180,E1 -7757.762,E2 -7757.762} C_VEL
LIN {X 0,Y 471.92,Z 537.791,A -85,B 0,C 180,E1 -7758.168,E2 -7758.168} C_VEL
LIN {X 0,Y 473.725,Z 416.336,A -85,B 0,C 180,E1 -7760.284,E2 -7760.284} C_VEL
LIN {X 0,Y 470.247,Z 397.717,A -85,B 0,C 180,E1 -7760.803,E2 -7760.803} C_VEL
LIN {X 0,Y 471.228,Z 378.492,A -85,B 0,C 180,E1 -7763.746,E2 -7763.746} C_VEL
LIN {X 0,Y 471.897,Z 366.725,A -85,B 0,C 180,E1 -7765.588,E2 -7765.588} C_VEL
LIN {X 0,Y 471.055,Z 361.57,A -85,B 0,C 180,E1 -7766.468,E2 -7766.468} C_VEL
LIN {X 0,Y 467.62,Z 347.314,A -85,B 0,C 180,E1 -7769.026,E2 -7769.026} C_VEL
LIN {X 0,Y 467.527,Z 346.873,A -85,B 0,C 180,E1 -7769.323,E2 -7769.323} C_VEL
LIN {X 0,Y 467.548,Z 346.871,A -85,B 0,C 180,E1 -7772.672,E2 -7772.672} C_VEL
LIN {X 0,Y 467.546,Z 346.873,A -85,B 0,C 180,E1 -7775.736,E2 -7775.736} C_VEL
LIN {X 0,Y 467.529,Z 346.87,A -85,B 0,C 180,E1 -7779.15,E2 -7779.15} C_VEL
LIN {X 0,Y 467.55,Z 346.867,A -85,B 0,C 180,E1 -7781.406,E2 -7781.406} C_VEL
LIN {X 0,Y 467.562,Z 346.867,A -85,B 0,C 180,E1 -7785.052,E2 -7785.052} C_VEL
LIN {X 0,Y 467.55,Z 346.869,A -85,B 0,C 180,E1 -7788.727,E2 -7788.727} C_VEL
LIN {X 0,Y 467.537,Z 346.875,A -85,B 0,C 180,E1 -7791.953,E2 -7791.953} C_VEL
LIN {X 0,Y 467.529,Z 346.872,A -85,B 0,C 180,E1 -7794.63,E2 -7794.63} C_VEL
LIN {X 0,Y 466.801,Z 347.013,A -85,B 0,C 180,E1 -7795.352,E2 -7795.352} C_VEL
LIN {X 0,Y 463.758,Z 347.346,A -85,B 0,C 180,E1 -7796.524,E2 -7796.524} C_VEL
LIN {X 0,Y 460.922,Z 347.694,A -85,B 0,C 180,E1 -7797.706,E2 -7797.706} C_VEL
LIN {X 0,Y 460.515,Z 347.842,A -85,B 0,C 180,E1 -7798.434,E2 -7798.434} C_VEL
LIN {X 0,Y 460.937,Z 349.621,A -85,B 0,C 180,E1 -7798.774,E2 -7798.774} C_VEL
LIN {X 0,Y 464.975,Z 365.295,A -85,B 0,C 180,E1 -7801.242,E2 -7801.242} C_VEL
LIN {X 0,Y 465.929,Z 369.718,A -85,B 0,C 180,E1 -7801.914,E2 -7801.914} C_VEL
LIN {X 0,Y 465.195,Z 388.983,A -85,B 0,C 180,E1 -7804.496,E2 -7804.496} C_VEL
LIN {X 0,Y 464.849,Z 397.492,A -85,B 0,C 180,E1 -7805.557,E2 -7805.557} C_VEL
LIN {X 0,Y 469.304,Z 420.448,A -85,B 0,C 180,E1 -7806.194,E2 -7806.194} C_VEL
LIN {X 0,Y 467.791,Z 553.35,A -85,B 0,C 180,E1 -7808.287,E2 -7808.287} C_VEL
LIN {X 0,Y 467.462,Z 570.388,A -85,B 0,C 180,E1 -7808.618,E2 -7808.618} C_VEL
LIN {X 0,Y 466.875,Z 585.583,A -85,B 0,C 180,E1 -7809.086,E2 -7809.086} C_VEL
LIN {X 0,Y 466.172,Z 600.133,A -85,B 0,C 180,E1 -7809.711,E2 -7809.711} C_VEL
LIN {X 0,Y 465.413,Z 613.937,A -85,B 0,C 180,E1 -7810.482,E2 -7810.482} C_VEL
LIN {X 0,Y 464.598,Z 626.685,A -85,B 0,C 180,E1 -7811.364,E2 -7811.364} C_VEL
LIN {X 0,Y 463.638,Z 639.847,A -85,B 0,C 180,E1 -7812.476,E2 -7812.476} C_VEL
LIN {X 0,Y 462.804,Z 651.682,A -85,B 0,C 180,E1 -7813.684,E2 -7813.684} C_VEL
LIN {X 0,Y 462.005,Z 662.601,A -85,B 0,C 180,E1 -7815.013,E2 -7815.013} C_VEL
LIN {X 0,Y 461.204,Z 673.201,A -85,B 0,C 180,E1 -7816.562,E2 -7816.562} C_VEL
LIN {X 0,Y 460.652,Z 682.029,A -85,B 0,C 180,E1 -7818.114,E2 -7818.114} C_VEL
LIN {X 0,Y 460.286,Z 688.364,A -85,B 0,C 180,E1 -7819.442,E2 -7819.442} C_VEL
LIN {X 0,Y 459.935,Z 695.376,A -85,B 0,C 180,E1 -7821.21,E2 -7821.21} C_VEL
LIN {X 0,Y 459.695,Z 700.895,A -85,B 0,C 180,E1 -7822.975,E2 -7822.975} C_VEL
LIN {X 0,Y 459.608,Z 705.073,A -85,B 0,C 180,E1 -7824.736,E2 -7824.736} C_VEL
LIN {X 0,Y 459.54,Z 708.01,A -85,B 0,C 180,E1 -7826.493,E2 -7826.493} C_VEL
LIN {X 0,Y 459.514,Z 709.773,A -85,B 0,C 180,E1 -7828.247,E2 -7828.247} C_VEL
LIN {X 0,Y 459.472,Z 710.385,A -85,B 0,C 180,E1 -7830,E2 -7830} C_VEL
LIN {X 0,Y 459.515,Z 709.819,A -85,B 0,C 180,E1 -7831.753,E2 -7831.753} C_VEL
LIN {X 0,Y 459.54,Z 708.12,A -85,B 0,C 180,E1 -7833.507,E2 -7833.507} C_VEL
LIN {X 0,Y 459.612,Z 705.253,A -85,B 0,C 180,E1 -7835.264,E2 -7835.264} C_VEL
LIN {X 0,Y 459.731,Z 701.15,A -85,B 0,C 180,E1 -7837.025,E2 -7837.025} C_VEL
LIN {X 0,Y 459.925,Z 695.702,A -85,B 0,C 180,E1 -7838.79,E2 -7838.79} C_VEL
LIN {X 0,Y 460.273,Z 688.763,A -85,B 0,C 180,E1 -7840.558,E2 -7840.558} C_VEL
LIN {X 0,Y 460.692,Z 681.337,A -85,B 0,C 180,E1 -7842.108,E2 -7842.108} C_VEL
LIN {X 0,Y 461.274,Z 672.391,A -85,B 0,C 180,E1 -7843.66,E2 -7843.66} C_VEL
LIN {X 0,Y 462.074,Z 661.583,A -85,B 0,C 180,E1 -7845.21,E2 -7845.21} C_VEL
LIN {X 0,Y 462.903,Z 650.492,A -85,B 0,C 180,E1 -7846.539,E2 -7846.539} C_VEL
LIN {X 0,Y 463.768,Z 638.328,A -85,B 0,C 180,E1 -7847.757,E2 -7847.757} C_VEL
LIN {X 0,Y 464.74,Z 624.919,A -85,B 0,C 180,E1 -7848.859,E2 -7848.859} C_VEL
LIN {X 0,Y 465.519,Z 611.832,A -85,B 0,C 180,E1 -7849.743,E2 -7849.743} C_VEL
LIN {X 0,Y 466.354,Z 597.51,A -85,B 0,C 180,E1 -7850.509,E2 -7850.509} C_VEL
LIN {X 0,Y 466.96,Z 582.721,A -85,B 0,C 180,E1 -7851.114,E2 -7851.114} C_VEL
LIN {X 0,Y 467.513,Z 567.293,A -85,B 0,C 180,E1 -7851.553,E2 -7851.553} C_VEL
LIN {X 0,Y 467.936,Z 537.611,A -85,B 0,C 180,E1 -7852.054,E2 -7852.054} C_VEL
LIN {X 0,Y 469.417,Z 421.465,A -85,B 0,C 180,E1 -7853.875,E2 -7853.875} C_VEL
LIN {X 0,Y 464.926,Z 397.33,A -85,B 0,C 180,E1 -7854.543,E2 -7854.543} C_VEL
LIN {X 0,Y 465.774,Z 375.4,A -85,B 0,C 180,E1 -7857.4,E2 -7857.4} C_VEL
LIN {X 0,Y 465.957,Z 370.349,A -85,B 0,C 180,E1 -7858.09,E2 -7858.09} C_VEL
LIN {X 0,Y 463.043,Z 357.583,A -85,B 0,C 180,E1 -7860.057,E2 -7860.057} C_VEL
LIN {X 0,Y 460.514,Z 347.873,A -85,B 0,C 180,E1 -7861.641,E2 -7861.641} C_VEL
LIN {X 0,Y 460.507,Z 347.75,A -85,B 0,C 180,E1 -7864.501,E2 -7864.501} C_VEL
LIN {X 0,Y 460.48,Z 347.753,A -85,B 0,C 180,E1 -7867.625,E2 -7867.625} C_VEL
LIN {X 0,Y 460.499,Z 347.746,A -85,B 0,C 180,E1 -7871.015,E2 -7871.015} C_VEL
LIN {X 0,Y 460.511,Z 347.743,A -85,B 0,C 180,E1 -7874.589,E2 -7874.589} C_VEL
LIN {X 0,Y 460.474,Z 347.751,A -85,B 0,C 180,E1 -7877.813,E2 -7877.813} C_VEL
LIN {X 0,Y 460.509,Z 347.745,A -85,B 0,C 180,E1 -7880.135,E2 -7880.135} C_VEL
LIN {X 0,Y 460.464,Z 347.755,A -85,B 0,C 180,E1 -7883.469,E2 -7883.469} C_VEL
LIN {X 0,Y 460.516,Z 347.743,A -85,B 0,C 180,E1 -7886.674,E2 -7886.674} C_VEL
LIN {X 0,Y 460.507,Z 347.747,A -85,B 0,C 180,E1 -7889.76,E2 -7889.76} C_VEL
LIN {X 0,Y 460.529,Z 347.734,A -85,B 0,C 180,E1 -7892.753,E2 -7892.753} C_VEL
LIN {X 0,Y 460.518,Z 347.748,A -85,B 0,C 180,E1 -7895.666,E2 -7895.666} C_VEL
LIN {X 0,Y 460.522,Z 347.737,A -85,B 0,C 180,E1 -7898.578,E2 -7898.578} C_VEL
LIN {X 0,Y 460.586,Z 347.738,A -85,B 0,C 180,E1 -7901.311,E2 -7901.311} C_VEL
LIN {X 0,Y 460.605,Z 347.73,A -85,B 0,C 180,E1 -7904.059,E2 -7904.059} C_VEL
LIN {X 0,Y 460.61,Z 347.729,A -85,B 0,C 180,E1 -7907.666,E2 -7907.666} C_VEL
LIN {X 0,Y 460.619,Z 347.731,A -85,B 0,C 180,E1 -7911.224,E2 -7911.224} C_VEL
LIN {X 0,Y 460.706,Z 347.714,A -85,B 0,C 180,E1 -7913.87,E2 -7913.87} C_VEL
LIN {X 0,Y 460.789,Z 347.711,A -85,B 0,C 180,E1 -7917.377,E2 -7917.377} C_VEL
LIN {X 0,Y 460.852,Z 347.696,A -85,B 0,C 180,E1 -7920,E2 -7920} C_VEL
LIN {X 0,Y 460.793,Z 347.701,A -85,B 0,C 180,E1 -7922.622,E2 -7922.622} C_VEL
LIN {X 0,Y 460.688,Z 347.717,A -85,B 0,C 180,E1 -7926.13,E2 -7926.13} C_VEL
LIN {X 0,Y 460.621,Z 347.721,A -85,B 0,C 180,E1 -7928.776,E2 -7928.776} C_VEL
LIN {X 0,Y 460.614,Z 347.726,A -85,B 0,C 180,E1 -7932.445,E2 -7932.445} C_VEL
LIN {X 0,Y 460.601,Z 347.732,A -85,B 0,C 180,E1 -7935.997,E2 -7935.997} C_VEL
LIN {X 0,Y 460.569,Z 347.73,A -85,B 0,C 180,E1 -7939.615,E2 -7939.615} C_VEL
LIN {X 0,Y 460.511,Z 347.744,A -85,B 0,C 180,E1 -7942.429,E2 -7942.429} C_VEL
LIN {X 0,Y 460.557,Z 347.736,A -85,B 0,C 180,E1 -7945.799,E2 -7945.799} C_VEL
LIN {X 0,Y 460.553,Z 347.738,A -85,B 0,C 180,E1 -7948.233,E2 -7948.233} C_VEL
LIN {X 0,Y 460.521,Z 347.747,A -85,B 0,C 180,E1 -7951.283,E2 -7951.283} C_VEL
LIN {X 0,Y 460.531,Z 347.737,A -85,B 0,C 180,E1 -7954.505,E2 -7954.505} C_VEL
LIN {X 0,Y 460.501,Z 347.742,A -85,B 0,C 180,E1 -7957.623,E2 -7957.623} C_VEL
LIN {X 0,Y 460.539,Z 347.715,A -85,B 0,C 180,E1 -7960.269,E2 -7960.269} C_VEL
LIN {X 0,Y 460.508,Z 347.748,A -85,B 0,C 180,E1 -7963.374,E2 -7963.374} C_VEL
LIN {X 0,Y 460.497,Z 347.73,A -85,B 0,C 180,E1 -7966.624,E2 -7966.624} C_VEL
LIN {X 0,Y 460.542,Z 347.741,A -85,B 0,C 180,E1 -7969.731,E2 -7969.731} C_VEL
LIN {X 0,Y 460.5,Z 347.75,A -85,B 0,C 180,E1 -7972.524,E2 -7972.524} C_VEL
LIN {X 0,Y 460.546,Z 347.744,A -85,B 0,C 180,E1 -7975.624,E2 -7975.624} C_VEL
LIN {X 0,Y 460.582,Z 347.952,A -85,B 0,C 180,E1 -7978.662,E2 -7978.662} C_VEL
LIN {X 0,Y 465.356,Z 365.725,A -85,B 0,C 180,E1 -7981.48,E2 -7981.48} C_VEL
LIN {X 0,Y 466.706,Z 371.573,A -85,B 0,C 180,E1 -7982.361,E2 -7982.361} C_VEL
LIN {X 0,Y 465.452,Z 391.627,A -85,B 0,C 180,E1 -7984.99,E2 -7984.99} C_VEL
LIN {X 0,Y 465.106,Z 398.228,A -85,B 0,C 180,E1 -7985.801,E2 -7985.801} C_VEL
LIN {X 0,Y 468.69,Z 419.558,A -85,B 0,C 180,E1 -7986.368,E2 -7986.368} C_VEL
LIN {X 0,Y 466.93,Z 565.708,A -85,B 0,C 180,E1 -7988.679,E2 -7988.679} C_VEL
LIN {X 0,Y 466.449,Z 581.493,A -85,B 0,C 180,E1 -7989.118,E2 -7989.118} C_VEL
LIN {X 0,Y 465.927,Z 594.795,A -85,B 0,C 180,E1 -7989.645,E2 -7989.645} C_VEL
LIN {X 0,Y 465.155,Z 608.638,A -85,B 0,C 180,E1 -7990.356,E2 -7990.356} C_VEL
LIN {X 0,Y 464.361,Z 622.215,A -85,B 0,C 180,E1 -7991.24,E2 -7991.24} C_VEL
LIN {X 0,Y 463.516,Z 634.684,A -85,B 0,C 180,E1 -7992.233,E2 -7992.233} C_VEL
LIN {X 0,Y 462.687,Z 647.3,A -85,B 0,C 180,E1 -7993.453,E2 -7993.453} C_VEL
LIN {X 0,Y 461.862,Z 658.726,A -85,B 0,C 180,E1 -7994.782,E2 -7994.782} C_VEL
LIN {X 0,Y 461.243,Z 668.324,A -85,B 0,C 180,E1 -7996.115,E2 -7996.115} C_VEL
LIN {X 0,Y 460.6,Z 677.723,A -85,B 0,C 180,E1 -7997.666,E2 -7997.666} C_VEL
LIN {X 0,Y 460.282,Z 685.525,A -85,B 0,C 180,E1 -7999.22,E2 -7999.22} C_VEL
LIN {X 0,Y 459.953,Z 691.99,A -85,B 0,C 180,E1 -8000.768,E2 -8000.768} C_VEL
LIN {X 0,Y 459.762,Z 697.912,A -85,B 0,C 180,E1 -8002.534,E2 -8002.534} C_VEL
LIN {X 0,Y 459.637,Z 701.405,A -85,B 0,C 180,E1 -8003.856,E2 -8003.856} C_VEL
LIN {X 0,Y 459.533,Z 704.951,A -85,B 0,C 180,E1 -8005.614,E2 -8005.614} C_VEL
LIN {X 0,Y 459.592,Z 707.284,A -85,B 0,C 180,E1 -8007.371,E2 -8007.371} C_VEL
LIN {X 0,Y 459.493,Z 708.459,A -85,B 0,C 180,E1 -8009.124,E2 -8009.124} C_VEL
LIN {X 0,Y 459.493,Z 708.46,A -85,B 0,C 180,E1 -8010.876,E2 -8010.876} C_VEL
LIN {X 0,Y 459.6,Z 707.288,A -85,B 0,C 180,E1 -8012.629,E2 -8012.629} C_VEL
LIN {X 0,Y 459.534,Z 704.954,A -85,B 0,C 180,E1 -8014.386,E2 -8014.386} C_VEL
LIN {X 0,Y 459.617,Z 701.402,A -85,B 0,C 180,E1 -8016.145,E2 -8016.145} C_VEL
LIN {X 0,Y 459.798,Z 696.549,A -85,B 0,C 180,E1 -8017.907,E2 -8017.907} C_VEL
LIN {X 0,Y 460.016,Z 690.267,A -85,B 0,C 180,E1 -8019.675,E2 -8019.675} C_VEL
LIN {X 0,Y 460.447,Z 682.362,A -85,B 0,C 180,E1 -8021.445,E2 -8021.445} C_VEL
LIN {X 0,Y 460.914,Z 674.047,A -85,B 0,C 180,E1 -8022.975,E2 -8022.975} C_VEL
LIN {X 0,Y 461.471,Z 665.336,A -85,B 0,C 180,E1 -8024.329,E2 -8024.329} C_VEL
LIN {X 0,Y 462.09,Z 655.163,A -85,B 0,C 180,E1 -8025.662,E2 -8025.662} C_VEL
LIN {X 0,Y 463.033,Z 642.741,A -85,B 0,C 180,E1 -8027.016,E2 -8027.016} C_VEL
LIN {X 0,Y 463.898,Z 629.434,A -85,B 0,C 180,E1 -8028.208,E2 -8028.208} C_VEL
LIN {X 0,Y 464.794,Z 615.785,A -85,B 0,C 180,E1 -8029.201,E2 -8029.201} C_VEL
LIN {X 0,Y 465.605,Z 601.544,A -85,B 0,C 180,E1 -8030.027,E2 -8030.027} C_VEL
LIN {X 0,Y 466.239,Z 587.009,A -85,B 0,C 180,E1 -8030.679,E2 -8030.679} C_VEL
LIN {X 0,Y 466.766,Z 572.5,A -85,B 0,C 180,E1 -8031.152,E2 -8031.152} C_VEL
LIN {X 0,Y 467.107,Z 556.546,A -85,B 0,C 180,E1 -8031.486,E2 -8031.486} C_VEL
LIN {X 0,Y 468.674,Z 426.809,A -85,B 0,C 180,E1 -8033.537,E2 -8033.537} C_VEL
LIN {X 0,Y 468.702,Z 418.361,A -85,B 0,C 180,E1 -8033.708,E2 -8033.708} C_VEL
LIN {X 0,Y 465.677,Z 399.731,A -85,B 0,C 180,E1 -8034.293,E2 -8034.293} C_VEL
LIN {X 0,Y 465.459,Z 398.259,A -85,B 0,C 180,E1 -8034.355,E2 -8034.355} C_VEL
LIN {X 0,Y 467.258,Z 377.044,A -85,B 0,C 180,E1 -8037.279,E2 -8037.279} C_VEL
LIN {X 0,Y 467.618,Z 373.593,A -85,B 0,C 180,E1 -8037.769,E2 -8037.769} C_VEL
LIN {X 0,Y 465.214,Z 362.977,A -85,B 0,C 180,E1 -8039.654,E2 -8039.654} C_VEL
LIN {X 0,Y 462.234,Z 353.178,A -85,B 0,C 180,E1 -8041.631,E2 -8041.631} C_VEL
LIN {X 0,Y 460.574,Z 347.854,A -85,B 0,C 180,E1 -8042.851,E2 -8042.851} C_VEL
LIN {X 0,Y 460.499,Z 347.75,A -85,B 0,C 180,E1 -8046.014,E2 -8046.014} C_VEL
LIN {X 0,Y 460.546,Z 347.745,A -85,B 0,C 180,E1 -8048.898,E2 -8048.898} C_VEL
LIN {X 0,Y 460.524,Z 347.747,A -85,B 0,C 180,E1 -8052.182,E2 -8052.182} C_VEL
LIN {X 0,Y 460.513,Z 347.747,A -85,B 0,C 180,E1 -8055.411,E2 -8055.411} C_VEL
LIN {X 0,Y 460.528,Z 347.746,A -85,B 0,C 180,E1 -8058.989,E2 -8058.989} C_VEL
LIN {X 0,Y 460.517,Z 347.748,A -85,B 0,C 180,E1 -8061.266,E2 -8061.266} C_VEL
LIN {X 0,Y 460.508,Z 347.751,A -85,B 0,C 180,E1 -8064.554,E2 -8064.554} C_VEL
LIN {X 0,Y 460.531,Z 347.746,A -85,B 0,C 180,E1 -8067.716,E2 -8067.716} C_VEL
LIN {X 0,Y 460.557,Z 348.001,A -85,B 0,C 180,E1 -8068.799,E2 -8068.799} C_VEL
LIN {X 0,Y 463.233,Z 356.896,A -85,B 0,C 180,E1 -8070.955,E2 -8070.955} C_VEL
LIN {X 0,Y 465.794,Z 367.412,A -85,B 0,C 180,E1 -8073.215,E2 -8073.215} C_VEL
LIN {X 0,Y 466.437,Z 371.904,A -85,B 0,C 180,E1 -8074.09,E2 -8074.09} C_VEL
LIN {X 0,Y 464.591,Z 393.86,A -85,B 0,C 180,E1 -8077.779,E2 -8077.779} C_VEL
LIN {X 0,Y 464.309,Z 398.291,A -85,B 0,C 180,E1 -8078.466,E2 -8078.466} C_VEL
LIN {X 0,Y 467.365,Z 412.97,A -85,B 0,C 180,E1 -8079.021,E2 -8079.021} C_VEL
LIN {X 0,Y 468.271,Z 418.356,A -85,B 0,C 180,E1 -8079.199,E2 -8079.199} C_VEL
LIN {X 0,Y 466.021,Z 504.725,A -85,B 0,C 180,E1 -8080.938,E2 -8080.938} C_VEL
LIN {X 0,Y 465.276,Z 541.521,A -85,B 0,C 180,E1 -8081.677,E2 -8081.677} C_VEL
LIN {X 0,Y 464.754,Z 556.861,A -85,B 0,C 180,E1 -8082.176,E2 -8082.176} C_VEL
LIN {X 0,Y 464.261,Z 570.824,A -85,B 0,C 180,E1 -8082.818,E2 -8082.818} C_VEL
LIN {X 0,Y 463.641,Z 583.984,A -85,B 0,C 180,E1 -8083.601,E2 -8083.601} C_VEL
LIN {X 0,Y 462.94,Z 597.166,A -85,B 0,C 180,E1 -8084.593,E2 -8084.593} C_VEL
LIN {X 0,Y 462.303,Z 609.044,A -85,B 0,C 180,E1 -8085.698,E2 -8085.698} C_VEL
LIN {X 0,Y 461.594,Z 620.668,A -85,B 0,C 180,E1 -8087.017,E2 -8087.017} C_VEL
LIN {X 0,Y 461.109,Z 630.274,A -85,B 0,C 180,E1 -8088.349,E2 -8088.349} C_VEL
LIN {X 0,Y 460.66,Z 638.174,A -85,B 0,C 180,E1 -8089.673,E2 -8089.673} C_VEL
LIN {X 0,Y 460.281,Z 645.738,A -85,B 0,C 180,E1 -8091.217,E2 -8091.217} C_VEL
LIN {X 0,Y 460.029,Z 650.964,A -85,B 0,C 180,E1 -8092.539,E2 -8092.539} C_VEL
LIN {X 0,Y 459.861,Z 656.434,A -85,B 0,C 180,E1 -8094.299,E2 -8094.299} C_VEL
LIN {X 0,Y 459.726,Z 659.437,A -85,B 0,C 180,E1 -8095.616,E2 -8095.616} C_VEL
LIN {X 0,Y 459.664,Z 662.198,A -85,B 0,C 180,E1 -8097.371,E2 -8097.371} C_VEL
LIN {X 0,Y 459.551,Z 663.558,A -85,B 0,C 180,E1 -8099.124,E2 -8099.124} C_VEL
LIN {X 0,Y 459.551,Z 663.529,A -85,B 0,C 180,E1 -8100.876,E2 -8100.876} C_VEL
LIN {X 0,Y 459.642,Z 662.105,A -85,B 0,C 180,E1 -8102.629,E2 -8102.629} C_VEL
LIN {X 0,Y 459.689,Z 659.275,A -85,B 0,C 180,E1 -8104.384,E2 -8104.384} C_VEL
LIN {X 0,Y 459.884,Z 654.963,A -85,B 0,C 180,E1 -8106.141,E2 -8106.141} C_VEL
LIN {X 0,Y 460.017,Z 649.054,A -85,B 0,C 180,E1 -8107.903,E2 -8107.903} C_VEL
LIN {X 0,Y 460.353,Z 642.383,A -85,B 0,C 180,E1 -8109.446,E2 -8109.446} C_VEL
LIN {X 0,Y 460.73,Z 634.096,A -85,B 0,C 180,E1 -8110.992,E2 -8110.992} C_VEL
LIN {X 0,Y 461.292,Z 625.411,A -85,B 0,C 180,E1 -8112.316,E2 -8112.316} C_VEL
LIN {X 0,Y 461.759,Z 614.881,A -85,B 0,C 180,E1 -8113.645,E2 -8113.645} C_VEL
LIN {X 0,Y 462.47,Z 603.112,A -85,B 0,C 180,E1 -8114.859,E2 -8114.859} C_VEL
LIN {X 0,Y 463.089,Z 591.388,A -85,B 0,C 180,E1 -8115.853,E2 -8115.853} C_VEL
LIN {X 0,Y 463.71,Z 578.558,A -85,B 0,C 180,E1 -8116.736,E2 -8116.736} C_VEL
LIN {X 0,Y 464.322,Z 565.27,A -85,B 0,C 180,E1 -8117.456,E2 -8117.456} C_VEL
LIN {X 0,Y 464.782,Z 551.294,A -85,B 0,C 180,E1 -8118.03,E2 -8118.03} C_VEL
LIN {X 0,Y 465.144,Z 536.651,A -85,B 0,C 180,E1 -8118.443,E2 -8118.443} C_VEL
LIN {X 0,Y 467.093,Z 418.059,A -85,B 0,C 180,E1 -8120.552,E2 -8120.552} C_VEL
LIN {X 0,Y 463.437,Z 398.005,A -85,B 0,C 180,E1 -8121.113,E2 -8121.113} C_VEL
LIN {X 0,Y 463.43,Z 396.113,A -85,B 0,C 180,E1 -8121.344,E2 -8121.344} C_VEL
LIN {X 0,Y 464.506,Z 377.326,A -85,B 0,C 180,E1 -8124.294,E2 -8124.294} C_VEL
LIN {X 0,Y 465.071,Z 368.143,A -85,B 0,C 180,E1 -8125.751,E2 -8125.751} C_VEL
LIN {X 0,Y 463.608,Z 360.707,A -85,B 0,C 180,E1 -8127.051,E2 -8127.051} C_VEL
LIN {X 0,Y 460.555,Z 348.171,A -85,B 0,C 180,E1 -8129.344,E2 -8129.344} C_VEL
LIN {X 0,Y 460.493,Z 347.763,A -85,B 0,C 180,E1 -8129.549,E2 -8129.549} C_VEL
LIN {X 0,Y 460.498,Z 347.751,A -85,B 0,C 180,E1 -8132.287,E2 -8132.287} C_VEL
LIN {X 0,Y 460.495,Z 347.749,A -85,B 0,C 180,E1 -8135.447,E2 -8135.447} C_VEL
LIN {X 0,Y 460.482,Z 347.748,A -85,B 0,C 180,E1 -8138.888,E2 -8138.888} C_VEL
LIN {X 0,Y 460.495,Z 347.746,A -85,B 0,C 180,E1 -8141.597,E2 -8141.597} C_VEL
LIN {X 0,Y 460.51,Z 347.747,A -85,B 0,C 180,E1 -8144.59,E2 -8144.59} C_VEL
LIN {X 0,Y 460.471,Z 347.745,A -85,B 0,C 180,E1 -8147.813,E2 -8147.813} C_VEL
LIN {X 0,Y 460.482,Z 347.746,A -85,B 0,C 180,E1 -8151.112,E2 -8151.112} C_VEL
LIN {X 0,Y 460.495,Z 347.75,A -85,B 0,C 180,E1 -8154.553,E2 -8154.553} C_VEL
LIN {X 0,Y 460.498,Z 347.746,A -85,B 0,C 180,E1 -8157.713,E2 -8157.713} C_VEL
LIN {X 0,Y 460.515,Z 347.842,A -85,B 0,C 180,E1 -8158.434,E2 -8158.434} C_VEL
LIN {X 0,Y 460.611,Z 349.207,A -85,B 0,C 180,E1 -8158.695,E2 -8158.695} C_VEL
LIN {X 0,Y 460.334,Z 353.639,A -85,B 0,C 180,E1 -8159.306,E2 -8159.306} C_VEL
LIN {X 0,Y 458.351,Z 365.434,A -85,B 0,C 180,E1 -8160.822,E2 -8160.822} C_VEL
LIN {X 0,Y 458.593,Z 368.962,A -85,B 0,C 180,E1 -8161.358,E2 -8161.358} C_VEL
LIN {X 0,Y 459.245,Z 372.755,A -85,B 0,C 180,E1 -8161.928,E2 -8161.928} C_VEL
LIN {X 0,Y 458.312,Z 392.512,A -85,B 0,C 180,E1 -8164.572,E2 -8164.572} C_VEL
LIN {X 0,Y 458.111,Z 397.315,A -85,B 0,C 180,E1 -8165.167,E2 -8165.167} C_VEL
LIN {X 0,Y 462.585,Z 420.429,A -85,B 0,C 180,E1 -8165.828,E2 -8165.828} C_VEL
LIN {X 0,Y 462.879,Z 425.043,A -85,B 0,C 180,E1 -8165.921,E2 -8165.921} C_VEL
LIN {X 0,Y 461.067,Z 564.253,A -85,B 0,C 180,E1 -8168.159,E2 -8168.159} C_VEL
LIN {X 0,Y 460.486,Z 579.462,A -85,B 0,C 180,E1 -8168.558,E2 -8168.558} C_VEL
LIN {X 0,Y 459.909,Z 593.562,A -85,B 0,C 180,E1 -8169.1,E2 -8169.1} C_VEL
LIN {X 0,Y 459.171,Z 606.435,A -85,B 0,C 180,E1 -8169.739,E2 -8169.739} C_VEL
LIN {X 0,Y 458.232,Z 620.589,A -85,B 0,C 180,E1 -8170.63,E2 -8170.63} C_VEL
LIN {X 0,Y 457.343,Z 633.501,A -85,B 0,C 180,E1 -8171.638,E2 -8171.638} C_VEL
LIN {X 0,Y 456.37,Z 646.281,A -85,B 0,C 180,E1 -8172.849,E2 -8172.849} C_VEL
LIN {X 0,Y 455.499,Z 657.356,A -85,B 0,C 180,E1 -8174.105,E2 -8174.105} C_VEL
LIN {X 0,Y 454.735,Z 667.381,A -85,B 0,C 180,E1 -8175.455,E2 -8175.455} C_VEL
LIN {X 0,Y 453.972,Z 677.432,A -85,B 0,C 180,E1 -8177.073,E2 -8177.073} C_VEL
LIN {X 0,Y 453.518,Z 685.315,A -85,B 0,C 180,E1 -8178.604,E2 -8178.604} C_VEL
LIN {X 0,Y 453.03,Z 692.054,A -85,B 0,C 180,E1 -8180.174,E2 -8180.174} C_VEL
LIN {X 0,Y 452.744,Z 698.297,A -85,B 0,C 180,E1 -8181.969,E2 -8181.969} C_VEL
LIN {X 0,Y 452.563,Z 703.13,A -85,B 0,C 180,E1 -8183.759,E2 -8183.759} C_VEL
LIN {X 0,Y 452.454,Z 706.679,A -85,B 0,C 180,E1 -8185.545,E2 -8185.545} C_VEL
LIN {X 0,Y 452.485,Z 709.022,A -85,B 0,C 180,E1 -8187.329,E2 -8187.329} C_VEL
LIN {X 0,Y 452.4,Z 710.214,A -85,B 0,C 180,E1 -8189.11,E2 -8189.11} C_VEL
LIN {X 0,Y 452.401,Z 710.229,A -85,B 0,C 180,E1 -8190.89,E2 -8190.89} C_VEL
LIN {X 0,Y 452.485,Z 709.098,A -85,B 0,C 180,E1 -8192.671,E2 -8192.671} C_VEL
LIN {X 0,Y 452.454,Z 706.82,A -85,B 0,C 180,E1 -8194.454,E2 -8194.454} C_VEL
LIN {X 0,Y 452.606,Z 702.99,A -85,B 0,C 180,E1 -8196.392,E2 -8196.392} C_VEL
LIN {X 0,Y 452.739,Z 698.586,A -85,B 0,C 180,E1 -8198.031,E2 -8198.031} C_VEL
LIN {X 0,Y 453.007,Z 692.412,A -85,B 0,C 180,E1 -8199.826,E2 -8199.826} C_VEL
LIN {X 0,Y 453.585,Z 684.653,A -85,B 0,C 180,E1 -8201.62,E2 -8201.62} C_VEL
LIN {X 0,Y 454.013,Z 676.518,A -85,B 0,C 180,E1 -8203.176,E2 -8203.176} C_VEL
LIN {X 0,Y 454.679,Z 667.985,A -85,B 0,C 180,E1 -8204.547,E2 -8204.547} C_VEL
LIN {X 0,Y 455.537,Z 656.258,A -85,B 0,C 180,E1 -8206.123,E2 -8206.123} C_VEL
LIN {X 0,Y 456.514,Z 644.15,A -85,B 0,C 180,E1 -8207.464,E2 -8207.464} C_VEL
LIN {X 0,Y 457.444,Z 631.932,A -85,B 0,C 180,E1 -8208.59,E2 -8208.59} C_VEL
LIN {X 0,Y 458.395,Z 618.677,A -85,B 0,C 180,E1 -8209.596,E2 -8209.596} C_VEL
LIN {X 0,Y 459.286,Z 605.055,A -85,B 0,C 180,E1 -8210.431,E2 -8210.431} C_VEL
LIN {X 0,Y 460.025,Z 590.141,A -85,B 0,C 180,E1 -8211.146,E2 -8211.146} C_VEL
LIN {X 0,Y 460.685,Z 575.691,A -85,B 0,C 180,E1 -8211.653,E2 -8211.653} C_VEL
LIN {X 0,Y 461.108,Z 560.387,A -85,B 0,C 180,E1 -8212.015,E2 -8212.015} C_VEL
LIN {X 0,Y 462.87,Z 421.957,A -85,B 0,C 180,E1 -8214.224,E2 -8214.224} C_VEL
LIN {X 0,Y 458.192,Z 397.293,A -85,B 0,C 180,E1 -8214.924,E2 -8214.924} C_VEL
LIN {X 0,Y 459.019,Z 376.954,A -85,B 0,C 180,E1 -8217.591,E2 -8217.591} C_VEL
LIN {X 0,Y 459.115,Z 371.623,A -85,B 0,C 180,E1 -8218.329,E2 -8218.329} C_VEL
LIN {X 0,Y 456.492,Z 360.306,A -85,B 0,C 180,E1 -8220.101,E2 -8220.101} C_VEL
LIN {X 0,Y 453.47,Z 348.759,A -85,B 0,C 180,E1 -8221.995,E2 -8221.995} C_VEL
LIN {X 0,Y 453.465,Z 348.626,A -85,B 0,C 180,E1 -8224.99,E2 -8224.99} C_VEL
LIN {X 0,Y 453.439,Z 348.626,A -85,B 0,C 180,E1 -8228.314,E2 -8228.314} C_VEL
LIN {X 0,Y 453.463,Z 348.623,A -85,B 0,C 180,E1 -8230.612,E2 -8230.612} C_VEL
LIN {X 0,Y 453.481,Z 348.619,A -85,B 0,C 180,E1 -8234.528,E2 -8234.528} C_VEL
LIN {X 0,Y 453.435,Z 348.628,A -85,B 0,C 180,E1 -8238.071,E2 -8238.071} C_VEL
LIN {X 0,Y 453.438,Z 348.622,A -85,B 0,C 180,E1 -8240.802,E2 -8240.802} C_VEL
LIN {X 0,Y 453.446,Z 348.623,A -85,B 0,C 180,E1 -8243.916,E2 -8243.916} C_VEL
LIN {X 0,Y 453.475,Z 348.622,A -85,B 0,C 180,E1 -8247.15,E2 -8247.15} C_VEL
LIN {X 0,Y 453.467,Z 348.623,A -85,B 0,C 180,E1 -8250.268,E2 -8250.268} C_VEL
LIN {X 0,Y 453.462,Z 348.616,A -85,B 0,C 180,E1 -8253.291,E2 -8253.291} C_VEL
LIN {X 0,Y 453.493,Z 348.616,A -85,B 0,C 180,E1 -8256.238,E2 -8256.238} C_VEL
LIN {X 0,Y 453.483,Z 348.615,A -85,B 0,C 180,E1 -8259.118,E2 -8259.118} C_VEL
LIN {X 0,Y 453.502,Z 348.613,A -85,B 0,C 180,E1 -8261.944,E2 -8261.944} C_VEL
LIN {X 0,Y 453.54,Z 348.608,A -85,B 0,C 180,E1 -8264.726,E2 -8264.726} C_VEL
LIN {X 0,Y 453.559,Z 348.601,A -85,B 0,C 180,E1 -8268.379,E2 -8268.379} C_VEL
LIN {X 0,Y 453.585,Z 348.605,A -85,B 0,C 180,E1 -8271.086,E2 -8271.086} C_VEL
LIN {X 0,Y 453.673,Z 348.591,A -85,B 0,C 180,E1 -8273.775,E2 -8273.775} C_VEL
LIN {X 0,Y 453.733,Z 348.589,A -85,B 0,C 180,E1 -8277.337,E2 -8277.337} C_VEL
LIN {X 0,Y 453.822,Z 348.572,A -85,B 0,C 180,E1 -8280,E2 -8280} C_VEL
LIN {X 0,Y 453.737,Z 348.58,A -85,B 0,C 180,E1 -8282.663,E2 -8282.663} C_VEL
LIN {X 0,Y 453.654,Z 348.593,A -85,B 0,C 180,E1 -8286.226,E2 -8286.226} C_VEL
LIN {X 0,Y 453.587,Z 348.598,A -85,B 0,C 180,E1 -8288.913,E2 -8288.913} C_VEL
LIN {X 0,Y 453.564,Z 348.605,A -85,B 0,C 180,E1 -8292.529,E2 -8292.529} C_VEL
LIN {X 0,Y 453.545,Z 348.61,A -85,B 0,C 180,E1 -8296.196,E2 -8296.196} C_VEL
LIN {X 0,Y 453.518,Z 348.611,A -85,B 0,C 180,E1 -8299.039,E2 -8299.039} C_VEL
LIN {X 0,Y 453.477,Z 348.621,A -85,B 0,C 180,E1 -8301.836,E2 -8301.836} C_VEL
LIN {X 0,Y 453.506,Z 348.612,A -85,B 0,C 180,E1 -8304.735,E2 -8304.735} C_VEL
LIN {X 0,Y 453.533,Z 348.613,A -85,B 0,C 180,E1 -8307.96,E2 -8307.96} C_VEL
LIN {X 0,Y 453.466,Z 348.625,A -85,B 0,C 180,E1 -8311.525,E2 -8311.525} C_VEL
LIN {X 0,Y 453.487,Z 348.615,A -85,B 0,C 180,E1 -8314.777,E2 -8314.777} C_VEL
LIN {X 0,Y 453.46,Z 348.618,A -85,B 0,C 180,E1 -8318.312,E2 -8318.312} C_VEL
LIN {X 0,Y 453.493,Z 348.593,A -85,B 0,C 180,E1 -8320.609,E2 -8320.609} C_VEL
LIN {X 0,Y 453.463,Z 348.628,A -85,B 0,C 180,E1 -8323.245,E2 -8323.245} C_VEL
LIN {X 0,Y 453.464,Z 348.61,A -85,B 0,C 180,E1 -8325.779,E2 -8325.779} C_VEL
LIN {X 0,Y 453.479,Z 348.614,A -85,B 0,C 180,E1 -8328.209,E2 -8328.209} C_VEL
LIN {X 0,Y 453.51,Z 348.622,A -85,B 0,C 180,E1 -8330.791,E2 -8330.791} C_VEL
LIN {X 0,Y 453.454,Z 348.624,A -85,B 0,C 180,E1 -8333.917,E2 -8333.917} C_VEL
LIN {X 0,Y 453.483,Z 348.625,A -85,B 0,C 180,E1 -8337.151,E2 -8337.151} C_VEL
LIN {X 0,Y 453.564,Z 348.863,A -85,B 0,C 180,E1 -8338.315,E2 -8338.315} C_VEL
LIN {X 0,Y 458.015,Z 365.513,A -85,B 0,C 180,E1 -8341.002,E2 -8341.002} C_VEL
LIN {X 0,Y 459.856,Z 372.899,A -85,B 0,C 180,E1 -8342.14,E2 -8342.14} C_VEL
LIN {X 0,Y 459.778,Z 377.024,A -85,B 0,C 180,E1 -8342.705,E2 -8342.705} C_VEL
LIN {X 0,Y 458.364,Z 397.716,A -85,B 0,C 180,E1 -8345.412,E2 -8345.412} C_VEL
LIN {X 0,Y 462.156,Z 419.889,A -85,B 0,C 180,E1 -8346.016,E2 -8346.016} C_VEL
LIN {X 0,Y 460.355,Z 564.446,A -85,B 0,C 180,E1 -8348.33,E2 -8348.33} C_VEL
LIN {X 0,Y 459.886,Z 580.271,A -85,B 0,C 180,E1 -8348.758,E2 -8348.758} C_VEL
LIN {X 0,Y 459.301,Z 593.826,A -85,B 0,C 180,E1 -8349.291,E2 -8349.291} C_VEL
LIN {X 0,Y 458.59,Z 606.709,A -85,B 0,C 180,E1 -8349.946,E2 -8349.946} C_VEL
LIN {X 0,Y 457.72,Z 620.677,A -85,B 0,C 180,E1 -8350.841,E2 -8350.841} C_VEL
LIN {X 0,Y 456.827,Z 633.429,A -85,B 0,C 180,E1 -8351.848,E2 -8351.848} C_VEL
LIN {X 0,Y 455.923,Z 645.856,A -85,B 0,C 180,E1 -8353.041,E2 -8353.041} C_VEL
LIN {X 0,Y 455.126,Z 656.975,A -85,B 0,C 180,E1 -8354.322,E2 -8354.322} C_VEL
LIN {X 0,Y 454.393,Z 666.865,A -85,B 0,C 180,E1 -8355.672,E2 -8355.672} C_VEL
LIN {X 0,Y 453.795,Z 675.534,A -85,B 0,C 180,E1 -8357.068,E2 -8357.068} C_VEL
LIN {X 0,Y 453.312,Z 684.539,A -85,B 0,C 180,E1 -8358.826,E2 -8358.826} C_VEL
LIN {X 0,Y 452.886,Z 692.007,A -85,B 0,C 180,E1 -8360.622,E2 -8360.622} C_VEL
LIN {X 0,Y 452.687,Z 697.928,A -85,B 0,C 180,E1 -8362.417,E2 -8362.417} C_VEL
LIN {X 0,Y 452.562,Z 701.42,A -85,B 0,C 180,E1 -8363.759,E2 -8363.759} C_VEL
LIN {X 0,Y 452.453,Z 704.965,A -85,B 0,C 180,E1 -8365.546,E2 -8365.546} C_VEL
LIN {X 0,Y 452.513,Z 707.299,A -85,B 0,C 180,E1 -8367.33,E2 -8367.33} C_VEL
LIN {X 0,Y 452.402,Z 708.473,A -85,B 0,C 180,E1 -8369.11,E2 -8369.11} C_VEL
LIN {X 0,Y 452.402,Z 708.474,A -85,B 0,C 180,E1 -8370.89,E2 -8370.89} C_VEL
LIN {X 0,Y 452.52,Z 707.302,A -85,B 0,C 180,E1 -8372.671,E2 -8372.671} C_VEL
LIN {X 0,Y 452.454,Z 704.968,A -85,B 0,C 180,E1 -8374.455,E2 -8374.455} C_VEL
LIN {X 0,Y 452.552,Z 701.201,A -85,B 0,C 180,E1 -8376.332,E2 -8376.332} C_VEL
LIN {X 0,Y 452.721,Z 696.564,A -85,B 0,C 180,E1 -8378.031,E2 -8378.031} C_VEL
LIN {X 0,Y 452.95,Z 690.283,A -85,B 0,C 180,E1 -8379.827,E2 -8379.827} C_VEL
LIN {X 0,Y 453.433,Z 682.378,A -85,B 0,C 180,E1 -8381.624,E2 -8381.624} C_VEL
LIN {X 0,Y 453.943,Z 674.065,A -85,B 0,C 180,E1 -8383.178,E2 -8383.178} C_VEL
LIN {X 0,Y 454.535,Z 665.355,A -85,B 0,C 180,E1 -8384.552,E2 -8384.552} C_VEL
LIN {X 0,Y 455.221,Z 655.184,A -85,B 0,C 180,E1 -8385.905,E2 -8385.905} C_VEL
LIN {X 0,Y 456.15,Z 643.471,A -85,B 0,C 180,E1 -8387.206,E2 -8387.206} C_VEL
LIN {X 0,Y 457.025,Z 630.826,A -85,B 0,C 180,E1 -8388.376,E2 -8388.376} C_VEL
LIN {X 0,Y 457.988,Z 617.503,A -85,B 0,C 180,E1 -8389.381,E2 -8389.381} C_VEL
LIN {X 0,Y 458.877,Z 602.696,A -85,B 0,C 180,E1 -8390.275,E2 -8390.275} C_VEL
LIN {X 0,Y 459.575,Z 587.724,A -85,B 0,C 180,E1 -8390.967,E2 -8390.967} C_VEL
LIN {X 0,Y 460.167,Z 572.023,A -85,B 0,C 180,E1 -8391.485,E2 -8391.485} C_VEL
LIN {X 0,Y 460.525,Z 556.677,A -85,B 0,C 180,E1 -8391.809,E2 -8391.809} C_VEL
LIN {X 0,Y 462.121,Z 432.99,A -85,B 0,C 180,E1 -8393.793,E2 -8393.793} C_VEL
LIN {X 0,Y 462.324,Z 419.5,A -85,B 0,C 180,E1 -8394.072,E2 -8394.072} C_VEL
LIN {X 0,Y 459.574,Z 402.113,A -85,B 0,C 180,E1 -8394.63,E2 -8394.63} C_VEL
LIN {X 0,Y 458.894,Z 398.183,A -85,B 0,C 180,E1 -8394.8,E2 -8394.8} C_VEL
LIN {X 0,Y 460.953,Z 376.783,A -85,B 0,C 180,E1 -8397.834,E2 -8397.834} C_VEL
LIN {X 0,Y 460.828,Z 374.417,A -85,B 0,C 180,E1 -8398.215,E2 -8398.215} C_VEL
LIN {X 0,Y 458.322,Z 364.072,A -85,B 0,C 180,E1 -8400.145,E2 -8400.145} C_VEL
LIN {X 0,Y 455.438,Z 354.478,A -85,B 0,C 180,E1 -8402.19,E2 -8402.19} C_VEL
LIN {X 0,Y 453.487,Z 348.714,A -85,B 0,C 180,E1 -8403.636,E2 -8403.636} C_VEL
LIN {X 0,Y 453.455,Z 348.628,A -85,B 0,C 180,E1 -8406.299,E2 -8406.299} C_VEL
LIN {X 0,Y 453.506,Z 348.622,A -85,B 0,C 180,E1 -8409.448,E2 -8409.448} C_VEL
LIN {X 0,Y 453.462,Z 348.628,A -85,B 0,C 180,E1 -8412.995,E2 -8412.995} C_VEL
LIN {X 0,Y 453.461,Z 348.626,A -85,B 0,C 180,E1 -8415.779,E2 -8415.779} C_VEL
LIN {X 0,Y 453.494,Z 348.622,A -85,B 0,C 180,E1 -8419.409,E2 -8419.409} C_VEL
LIN {X 0,Y 453.45,Z 348.629,A -85,B 0,C 180,E1 -8422.81,E2 -8422.81} C_VEL
LIN {X 0,Y 453.475,Z 348.627,A -85,B 0,C 180,E1 -8426.087,E2 -8426.087} C_VEL
LIN {X 0,Y 453.509,Z 348.826,A -85,B 0,C 180,E1 -8428.041,E2 -8428.041} C_VEL
LIN {X 0,Y 456.395,Z 358.303,A -85,B 0,C 180,E1 -8430.478,E2 -8430.478} C_VEL
LIN {X 0,Y 458.849,Z 368.026,A -85,B 0,C 180,E1 -8432.669,E2 -8432.669} C_VEL
LIN {X 0,Y 459.815,Z 372.921,A -85,B 0,C 180,E1 -8433.689,E2 -8433.689} C_VEL
LIN {X 0,Y 458.534,Z 387.827,A -85,B 0,C 180,E1 -8436.276,E2 -8436.276} C_VEL
LIN {X 0,Y 457.665,Z 398.271,A -85,B 0,C 180,E1 -8438.002,E2 -8438.002} C_VEL
LIN {X 0,Y 460.773,Z 412.495,A -85,B 0,C 180,E1 -8438.588,E2 -8438.588} C_VEL
LIN {X 0,Y 461.906,Z 420.304,A -85,B 0,C 180,E1 -8438.847,E2 -8438.847} C_VEL
LIN {X 0,Y 459.432,Z 505.607,A -85,B 0,C 180,E1 -8440.625,E2 -8440.625} C_VEL
LIN {X 0,Y 458.631,Z 541.65,A -85,B 0,C 180,E1 -8441.373,E2 -8441.373} C_VEL
LIN {X 0,Y 458.062,Z 557.237,A -85,B 0,C 180,E1 -8441.891,E2 -8441.891} C_VEL
LIN {X 0,Y 457.503,Z 571.878,A -85,B 0,C 180,E1 -8442.582,E2 -8442.582} C_VEL
LIN {X 0,Y 456.849,Z 584.468,A -85,B 0,C 180,E1 -8443.35,E2 -8443.35} C_VEL
LIN {X 0,Y 456.108,Z 597.595,A -85,B 0,C 180,E1 -8444.357,E2 -8444.357} C_VEL
LIN {X 0,Y 455.445,Z 609.442,A -85,B 0,C 180,E1 -8445.478,E2 -8445.478} C_VEL
LIN {X 0,Y 454.714,Z 620.435,A -85,B 0,C 180,E1 -8446.738,E2 -8446.738} C_VEL
LIN {X 0,Y 454.153,Z 630.656,A -85,B 0,C 180,E1 -8448.168,E2 -8448.168} C_VEL
LIN {X 0,Y 453.679,Z 638.555,A -85,B 0,C 180,E1 -8449.513,E2 -8449.513} C_VEL
LIN {X 0,Y 453.273,Z 646.122,A -85,B 0,C 180,E1 -8451.08,E2 -8451.08} C_VEL
LIN {X 0,Y 453.002,Z 651.346,A -85,B 0,C 180,E1 -8452.422,E2 -8452.422} C_VEL
LIN {X 0,Y 452.891,Z 655.57,A -85,B 0,C 180,E1 -8453.764,E2 -8453.764} C_VEL
LIN {X 0,Y 452.643,Z 659.817,A -85,B 0,C 180,E1 -8455.548,E2 -8455.548} C_VEL
LIN {X 0,Y 452.586,Z 662.57,A -85,B 0,C 180,E1 -8457.33,E2 -8457.33} C_VEL
LIN {X 0,Y 452.487,Z 663.916,A -85,B 0,C 180,E1 -8459.11,E2 -8459.11} C_VEL
LIN {X 0,Y 452.487,Z 663.864,A -85,B 0,C 180,E1 -8460.89,E2 -8460.89} C_VEL
LIN {X 0,Y 452.566,Z 662.413,A -85,B 0,C 180,E1 -8462.67,E2 -8462.67} C_VEL
LIN {X 0,Y 452.635,Z 661.159,A -85,B 0,C 180,E1 -8463.561,E2 -8463.561} C_VEL
LIN {X 0,Y 452.685,Z 657.566,A -85,B 0,C 180,E1 -8465.345,E2 -8465.345} C_VEL
LIN {X 0,Y 452.835,Z 654.02,A -85,B 0,C 180,E1 -8466.645,E2 -8466.645} C_VEL
LIN {X 0,Y 452.985,Z 649.242,A -85,B 0,C 180,E1 -8468.027,E2 -8468.027} C_VEL
LIN {X 0,Y 453.33,Z 642.52,A -85,B 0,C 180,E1 -8469.594,E2 -8469.594} C_VEL
LIN {X 0,Y 453.74,Z 634.162,A -85,B 0,C 180,E1 -8471.164,E2 -8471.164} C_VEL
LIN {X 0,Y 454.293,Z 625.407,A -85,B 0,C 180,E1 -8472.509,E2 -8472.509} C_VEL
LIN {X 0,Y 454.83,Z 614.785,A -85,B 0,C 180,E1 -8473.857,E2 -8473.857} C_VEL
LIN {X 0,Y 455.525,Z 602.922,A -85,B 0,C 180,E1 -8475.091,E2 -8475.091} C_VEL
LIN {X 0,Y 456.206,Z 591.09,A -85,B 0,C 180,E1 -8476.099,E2 -8476.099} C_VEL
LIN {X 0,Y 456.872,Z 578.128,A -85,B 0,C 180,E1 -8476.994,E2 -8476.994} C_VEL
LIN {X 0,Y 457.512,Z 564.196,A -85,B 0,C 180,E1 -8477.748,E2 -8477.748} C_VEL
LIN {X 0,Y 457.998,Z 550.361,A -85,B 0,C 180,E1 -8478.306,E2 -8478.306} C_VEL
LIN {X 0,Y 458.361,Z 536.413,A -85,B 0,C 180,E1 -8478.696,E2 -8478.696} C_VEL
LIN {X 0,Y 460.433,Z 418.974,A -85,B 0,C 180,E1 -8480.838,E2 -8480.838} C_VEL
LIN {X 0,Y 456.538,Z 397.59,A -85,B 0,C 180,E1 -8481.46,E2 -8481.46} C_VEL
LIN {X 0,Y 457.581,Z 379.857,A -85,B 0,C 180,E1 -8484.259,E2 -8484.259} C_VEL
LIN {X 0,Y 458.206,Z 369.512,A -85,B 0,C 180,E1 -8485.921,E2 -8485.921} C_VEL
LIN {X 0,Y 456.025,Z 359.331,A -85,B 0,C 180,E1 -8487.743,E2 -8487.743} C_VEL
LIN {X 0,Y 453.464,Z 348.821,A -85,B 0,C 180,E1 -8489.733,E2 -8489.733} C_VEL
LIN {X 0,Y 453.455,Z 348.626,A -85,B 0,C 180,E1 -8492.851,E2 -8492.851} C_VEL
LIN {X 0,Y 453.467,Z 348.623,A -85,B 0,C 180,E1 -8494.991,E2 -8494.991} C_VEL
LIN {X 0,Y 453.44,Z 348.629,A -85,B 0,C 180,E1 -8498.314,E2 -8498.314} C_VEL
LIN {X 0,Y 453.467,Z 348.622,A -85,B 0,C 180,E1 -8500.612,E2 -8500.612} C_VEL
LIN {X 0,Y 453.481,Z 348.623,A -85,B 0,C 180,E1 -8504.528,E2 -8504.528} C_VEL
LIN {X 0,Y 453.437,Z 348.627,A -85,B 0,C 180,E1 -8508.204,E2 -8508.204} C_VEL
LIN {X 0,Y 453.424,Z 348.624,A -85,B 0,C 180,E1 -8510.804,E2 -8510.804} C_VEL
LIN {X 0,Y 453.438,Z 348.624,A -85,B 0,C 180,E1 -8513.915,E2 -8513.915} C_VEL
LIN {X 0,Y 453.465,Z 348.627,A -85,B 0,C 180,E1 -8516.816,E2 -8516.816} C_VEL
LIN {X 0,Y 453.498,Z 348.852,A -85,B 0,C 180,E1 -8518.138,E2 -8518.138} C_VEL
LIN {X 0,Y 458.07,Z 366.569,A -85,B 0,C 180,E1 -8520.99,E2 -8520.99} C_VEL
LIN {X 0,Y 458.593,Z 368.962,A -85,B 0,C 180,E1 -8521.358,E2 -8521.358} C_VEL
LIN {X 0,Y 458.31,Z 371.634,A -85,B 0,C 180,E1 -8521.715,E2 -8521.715} C_VEL
LIN {X 0,Y 455.704,Z 376.353,A -85,B 0,C 180,E1 -8522.214,E2 -8522.214} C_VEL
LIN {X 0,Y 452.75,Z 381.183,A -85,B 0,C 180,E1 -8522.708,E2 -8522.708} C_VEL
LIN {X 0,Y 451.989,Z 384.049,A -85,B 0,C 180,E1 -8523.058,E2 -8523.058} C_VEL
LIN {X 0,Y 451.433,Z 397.229,A -85,B 0,C 180,E1 -8524.774,E2 -8524.774} C_VEL
LIN {X 0,Y 456.341,Z 422.736,A -85,B 0,C 180,E1 -8525.517,E2 -8525.517} C_VEL
LIN {X 0,Y 454.611,Z 554.895,A -85,B 0,C 180,E1 -8527.654,E2 -8527.654} C_VEL
LIN {X 0,Y 454.228,Z 571.296,A -85,B 0,C 180,E1 -8527.993,E2 -8527.993} C_VEL
LIN {X 0,Y 453.573,Z 586.349,A -85,B 0,C 180,E1 -8528.478,E2 -8528.478} C_VEL
LIN {X 0,Y 452.791,Z 601.144,A -85,B 0,C 180,E1 -8529.144,E2 -8529.144} C_VEL
LIN {X 0,Y 451.874,Z 615.588,A -85,B 0,C 180,E1 -8529.991,E2 -8529.991} C_VEL
LIN {X 0,Y 450.861,Z 629.411,A -85,B 0,C 180,E1 -8531.01,E2 -8531.01} C_VEL
LIN {X 0,Y 449.846,Z 642.118,A -85,B 0,C 180,E1 -8532.158,E2 -8532.158} C_VEL
LIN {X 0,Y 448.927,Z 653.557,A -85,B 0,C 180,E1 -8533.399,E2 -8533.399} C_VEL
LIN {X 0,Y 448.039,Z 664.165,A -85,B 0,C 180,E1 -8534.767,E2 -8534.767} C_VEL
LIN {X 0,Y 447.166,Z 674.5,A -85,B 0,C 180,E1 -8536.364,E2 -8536.364} C_VEL
LIN {X 0,Y 446.575,Z 683.121,A -85,B 0,C 180,E1 -8537.969,E2 -8537.969} C_VEL
LIN {X 0,Y 446.118,Z 690.255,A -85,B 0,C 180,E1 -8539.562,E2 -8539.562} C_VEL
LIN {X 0,Y 445.752,Z 696.878,A -85,B 0,C 180,E1 -8541.386,E2 -8541.386} C_VEL
LIN {X 0,Y 445.502,Z 702.063,A -85,B 0,C 180,E1 -8543.205,E2 -8543.205} C_VEL
LIN {X 0,Y 445.441,Z 705.046,A -85,B 0,C 180,E1 -8544.568,E2 -8544.568} C_VEL
LIN {X 0,Y 445.336,Z 707.983,A -85,B 0,C 180,E1 -8546.381,E2 -8546.381} C_VEL
LIN {X 0,Y 445.349,Z 709.746,A -85,B 0,C 180,E1 -8548.191,E2 -8548.191} C_VEL
LIN {X 0,Y 445.29,Z 710.357,A -85,B 0,C 180,E1 -8550,E2 -8550} C_VEL
LIN {X 0,Y 445.35,Z 709.791,A -85,B 0,C 180,E1 -8551.809,E2 -8551.809} C_VEL
LIN {X 0,Y 445.337,Z 708.09,A -85,B 0,C 180,E1 -8553.619,E2 -8553.619} C_VEL
LIN {X 0,Y 445.449,Z 705.222,A -85,B 0,C 180,E1 -8555.432,E2 -8555.432} C_VEL
LIN {X 0,Y 445.585,Z 701.117,A -85,B 0,C 180,E1 -8557.249,E2 -8557.249} C_VEL
LIN {X 0,Y 445.809,Z 695.667,A -85,B 0,C 180,E1 -8559.07,E2 -8559.07} C_VEL
LIN {X 0,Y 446.255,Z 688.725,A -85,B 0,C 180,E1 -8560.894,E2 -8560.894} C_VEL
LIN {X 0,Y 446.715,Z 680.935,A -85,B 0,C 180,E1 -8562.562,E2 -8562.562} C_VEL
LIN {X 0,Y 447.382,Z 672.346,A -85,B 0,C 180,E1 -8564.093,E2 -8564.093} C_VEL
LIN {X 0,Y 448.265,Z 661.531,A -85,B 0,C 180,E1 -8565.691,E2 -8565.691} C_VEL
LIN {X 0,Y 449.228,Z 650.434,A -85,B 0,C 180,E1 -8567.058,E2 -8567.058} C_VEL
LIN {X 0,Y 450.164,Z 638.261,A -85,B 0,C 180,E1 -8568.312,E2 -8568.312} C_VEL
LIN {X 0,Y 451.281,Z 624.841,A -85,B 0,C 180,E1 -8569.444,E2 -8569.444} C_VEL
LIN {X 0,Y 452.152,Z 611.738,A -85,B 0,C 180,E1 -8570.352,E2 -8570.352} C_VEL
LIN {X 0,Y 453.015,Z 598.022,A -85,B 0,C 180,E1 -8571.11,E2 -8571.11} C_VEL
LIN {X 0,Y 453.72,Z 583.127,A -85,B 0,C 180,E1 -8571.741,E2 -8571.741} C_VEL
LIN {X 0,Y 454.322,Z 568.271,A -85,B 0,C 180,E1 -8572.182,E2 -8572.182} C_VEL
LIN {X 0,Y 454.719,Z 546.183,A -85,B 0,C 180,E1 -8572.58,E2 -8572.58} C_VEL
LIN {X 0,Y 456.406,Z 423.087,A -85,B 0,C 180,E1 -8574.567,E2 -8574.567} C_VEL
LIN {X 0,Y 451.51,Z 397.546,A -85,B 0,C 180,E1 -8575.3,E2 -8575.3} C_VEL
LIN {X 0,Y 451.641,Z 391.272,A -85,B 0,C 180,E1 -8576.078,E2 -8576.078} C_VEL
LIN {X 0,Y 452.41,Z 374.922,A -85,B 0,C 180,E1 -8578.281,E2 -8578.281} C_VEL
LIN {X 0,Y 451.609,Z 369.883,A -85,B 0,C 180,E1 -8579.053,E2 -8579.053} C_VEL
LIN {X 0,Y 447.523,Z 353.672,A -85,B 0,C 180,E1 -8581.659,E2 -8581.659} C_VEL
LIN {X 0,Y 446.449,Z 349.647,A -85,B 0,C 180,E1 -8582.359,E2 -8582.359} C_VEL
LIN {X 0,Y 446.405,Z 349.498,A -85,B 0,C 180,E1 -8585.627,E2 -8585.627} C_VEL
LIN {X 0,Y 446.386,Z 349.498,A -85,B 0,C 180,E1 -8589.033,E2 -8589.033} C_VEL
LIN {X 0,Y 446.377,Z 349.505,A -85,B 0,C 180,E1 -8592.269,E2 -8592.269} C_VEL
LIN {X 0,Y 446.421,Z 349.498,A -85,B 0,C 180,E1 -8595.108,E2 -8595.108} C_VEL
LIN {X 0,Y 446.399,Z 349.504,A -85,B 0,C 180,E1 -8598.606,E2 -8598.606} C_VEL
LIN {X 0,Y 446.399,Z 349.506,A -85,B 0,C 180,E1 -8601.923,E2 -8601.923} C_VEL
LIN {X 0,Y 446.421,Z 349.498,A -85,B 0,C 180,E1 -8605.476,E2 -8605.476} C_VEL
LIN {X 0,Y 446.414,Z 349.493,A -85,B 0,C 180,E1 -8608.699,E2 -8608.699} C_VEL
LIN {X 0,Y 446.449,Z 349.493,A -85,B 0,C 180,E1 -8611.83,E2 -8611.83} C_VEL
LIN {X 0,Y 446.421,Z 349.499,A -85,B 0,C 180,E1 -8614.845,E2 -8614.845} C_VEL
LIN {X 0,Y 446.449,Z 349.491,A -85,B 0,C 180,E1 -8618.245,E2 -8618.245} C_VEL
LIN {X 0,Y 446.451,Z 349.495,A -85,B 0,C 180,E1 -8621.649,E2 -8621.649} C_VEL
LIN {X 0,Y 446.508,Z 349.484,A -85,B 0,C 180,E1 -8624.48,E2 -8624.48} C_VEL
LIN {X 0,Y 446.517,Z 349.478,A -85,B 0,C 180,E1 -8628.193,E2 -8628.193} C_VEL
LIN {X 0,Y 446.533,Z 349.482,A -85,B 0,C 180,E1 -8630.944,E2 -8630.944} C_VEL
LIN {X 0,Y 446.641,Z 349.468,A -85,B 0,C 180,E1 -8633.676,E2 -8633.676} C_VEL
LIN {X 0,Y 446.679,Z 349.467,A -85,B 0,C 180,E1 -8637.294,E2 -8637.294} C_VEL
LIN {X 0,Y 446.792,Z 349.447,A -85,B 0,C 180,E1 -8640,E2 -8640} C_VEL
LIN {X 0,Y 446.685,Z 349.459,A -85,B 0,C 180,E1 -8642.705,E2 -8642.705} C_VEL
LIN {X 0,Y 446.622,Z 349.469,A -85,B 0,C 180,E1 -8646.324,E2 -8646.324} C_VEL
LIN {X 0,Y 446.523,Z 349.485,A -85,B 0,C 180,E1 -8649.97,E2 -8649.97} C_VEL
LIN {X 0,Y 446.522,Z 349.483,A -85,B 0,C 180,E1 -8652.73,E2 -8652.73} C_VEL
LIN {X 0,Y 446.496,Z 349.488,A -85,B 0,C 180,E1 -8656.227,E2 -8656.227} C_VEL
LIN {X 0,Y 446.469,Z 349.486,A -85,B 0,C 180,E1 -8659.303,E2 -8659.303} C_VEL
LIN {X 0,Y 446.418,Z 349.499,A -85,B 0,C 180,E1 -8662.199,E2 -8662.199} C_VEL
LIN {X 0,Y 446.449,Z 349.49,A -85,B 0,C 180,E1 -8665.153,E2 -8665.153} C_VEL
LIN {X 0,Y 446.485,Z 349.491,A -85,B 0,C 180,E1 -8668.179,E2 -8668.179} C_VEL
LIN {X 0,Y 446.419,Z 349.501,A -85,B 0,C 180,E1 -8671.775,E2 -8671.775} C_VEL
LIN {X 0,Y 446.429,Z 349.493,A -85,B 0,C 180,E1 -8674.523,E2 -8674.523} C_VEL
LIN {X 0,Y 446.413,Z 349.495,A -85,B 0,C 180,E1 -8678.079,E2 -8678.079} C_VEL
LIN {X 0,Y 446.426,Z 349.474,A -85,B 0,C 180,E1 -8680.917,E2 -8680.917} C_VEL
LIN {X 0,Y 446.422,Z 349.5,A -85,B 0,C 180,E1 -8683.843,E2 -8683.843} C_VEL
LIN {X 0,Y 446.397,Z 349.485,A -85,B 0,C 180,E1 -8686.404,E2 -8686.404} C_VEL
LIN {X 0,Y 446.427,Z 349.503,A -85,B 0,C 180,E1 -8689.082,E2 -8689.082} C_VEL
LIN {X 0,Y 446.416,Z 349.502,A -85,B 0,C 180,E1 -8691.921,E2 -8691.921} C_VEL
LIN {X 0,Y 446.429,Z 349.502,A -85,B 0,C 180,E1 -8695.477,E2 -8695.477} C_VEL
LIN {X 0,Y 446.5,Z 349.677,A -85,B 0,C 180,E1 -8697.929,E2 -8697.929} C_VEL
LIN {X 0,Y 451.462,Z 368.251,A -85,B 0,C 180,E1 -8700.981,E2 -8700.981} C_VEL
LIN {X 0,Y 453.16,Z 375.643,A -85,B 0,C 180,E1 -8702.129,E2 -8702.129} C_VEL
LIN {X 0,Y 451.625,Z 397.191,A -85,B 0,C 180,E1 -8705.006,E2 -8705.006} C_VEL
LIN {X 0,Y 455.679,Z 420.944,A -85,B 0,C 180,E1 -8705.668,E2 -8705.668} C_VEL
LIN {X 0,Y 453.774,Z 564.578,A -85,B 0,C 180,E1 -8708,E2 -8708} C_VEL
LIN {X 0,Y 453.291,Z 580.048,A -85,B 0,C 180,E1 -8708.424,E2 -8708.424} C_VEL
LIN {X 0,Y 452.652,Z 594.133,A -85,B 0,C 180,E1 -8708.984,E2 -8708.984} C_VEL
LIN {X 0,Y 451.788,Z 608.728,A -85,B 0,C 180,E1 -8709.75,E2 -8709.75} C_VEL
LIN {X 0,Y 450.897,Z 622.289,A -85,B 0,C 180,E1 -8710.657,E2 -8710.657} C_VEL
LIN {X 0,Y 449.856,Z 636.033,A -85,B 0,C 180,E1 -8711.793,E2 -8711.793} C_VEL
LIN {X 0,Y 448.954,Z 648.112,A -85,B 0,C 180,E1 -8713.015,E2 -8713.015} C_VEL
LIN {X 0,Y 448.103,Z 658.774,A -85,B 0,C 180,E1 -8714.303,E2 -8714.303} C_VEL
LIN {X 0,Y 447.354,Z 668.368,A -85,B 0,C 180,E1 -8715.674,E2 -8715.674} C_VEL
LIN {X 0,Y 446.604,Z 678.086,A -85,B 0,C 180,E1 -8717.334,E2 -8717.334} C_VEL
LIN {X 0,Y 446.192,Z 686.566,A -85,B 0,C 180,E1 -8719.105,E2 -8719.105} C_VEL
LIN {X 0,Y 445.773,Z 693.633,A -85,B 0,C 180,E1 -8720.929,E2 -8720.929} C_VEL
LIN {X 0,Y 445.569,Z 699.182,A -85,B 0,C 180,E1 -8722.751,E2 -8722.751} C_VEL
LIN {X 0,Y 445.448,Z 703.364,A -85,B 0,C 180,E1 -8724.568,E2 -8724.568} C_VEL
LIN {X 0,Y 445.347,Z 706.294,A -85,B 0,C 180,E1 -8726.381,E2 -8726.381} C_VEL
LIN {X 0,Y 445.375,Z 708.043,A -85,B 0,C 180,E1 -8728.192,E2 -8728.192} C_VEL
LIN {X 0,Y 445.289,Z 708.64,A -85,B 0,C 180,E1 -8730,E2 -8730} C_VEL
LIN {X 0,Y 445.377,Z 708.044,A -85,B 0,C 180,E1 -8731.809,E2 -8731.809} C_VEL
LIN {X 0,Y 445.348,Z 706.297,A -85,B 0,C 180,E1 -8733.619,E2 -8733.619} C_VEL
LIN {X 0,Y 445.441,Z 703.363,A -85,B 0,C 180,E1 -8735.432,E2 -8735.432} C_VEL
LIN {X 0,Y 445.568,Z 699.174,A -85,B 0,C 180,E1 -8737.249,E2 -8737.249} C_VEL
LIN {X 0,Y 445.773,Z 693.627,A -85,B 0,C 180,E1 -8739.071,E2 -8739.071} C_VEL
LIN {X 0,Y 446.201,Z 686.564,A -85,B 0,C 180,E1 -8740.895,E2 -8740.895} C_VEL
LIN {X 0,Y 446.58,Z 679.048,A -85,B 0,C 180,E1 -8742.485,E2 -8742.485} C_VEL
LIN {X 0,Y 447.279,Z 669.833,A -85,B 0,C 180,E1 -8744.096,E2 -8744.096} C_VEL
LIN {X 0,Y 447.972,Z 660.509,A -85,B 0,C 180,E1 -8745.468,E2 -8745.468} C_VEL
LIN {X 0,Y 448.9,Z 648.5,A -85,B 0,C 180,E1 -8746.941,E2 -8746.941} C_VEL
LIN {X 0,Y 449.913,Z 635.993,A -85,B 0,C 180,E1 -8748.205,E2 -8748.205} C_VEL
LIN {X 0,Y 450.833,Z 623.807,A -85,B 0,C 180,E1 -8749.227,E2 -8749.227} C_VEL
LIN {X 0,Y 451.732,Z 610.58,A -85,B 0,C 180,E1 -8750.134,E2 -8750.134} C_VEL
LIN {X 0,Y 452.525,Z 596.013,A -85,B 0,C 180,E1 -8750.929,E2 -8750.929} C_VEL
LIN {X 0,Y 453.283,Z 580.455,A -85,B 0,C 180,E1 -8751.559,E2 -8751.559} C_VEL
LIN {X 0,Y 453.754,Z 565.792,A -85,B 0,C 180,E1 -8751.972,E2 -8751.972} C_VEL
LIN {X 0,Y 455.03,Z 472.509,A -85,B 0,C 180,E1 -8753.496,E2 -8753.496} C_VEL
LIN {X 0,Y 455.546,Z 441.129,A -85,B 0,C 180,E1 -8754.025,E2 -8754.025} C_VEL
LIN {X 0,Y 456,Z 420.479,A -85,B 0,C 180,E1 -8754.455,E2 -8754.455} C_VEL
LIN {X 0,Y 453.293,Z 403.198,A -85,B 0,C 180,E1 -8755.046,E2 -8755.046} C_VEL
LIN {X 0,Y 452.389,Z 398.189,A -85,B 0,C 180,E1 -8755.258,E2 -8755.258} C_VEL
LIN {X 0,Y 454.514,Z 378.035,A -85,B 0,C 180,E1 -8758.192,E2 -8758.192} C_VEL
LIN {X 0,Y 452.306,Z 368.205,A -85,B 0,C 180,E1 -8760.056,E2 -8760.056} C_VEL
LIN {X 0,Y 449.209,Z 357.702,A -85,B 0,C 180,E1 -8762.345,E2 -8762.345} C_VEL
LIN {X 0,Y 446.469,Z 349.718,A -85,B 0,C 180,E1 -8764.417,E2 -8764.417} C_VEL
LIN {X 0,Y 446.403,Z 349.507,A -85,B 0,C 180,E1 -8766.745,E2 -8766.745} C_VEL
LIN {X 0,Y 446.469,Z 349.498,A -85,B 0,C 180,E1 -8769.527,E2 -8769.527} C_VEL
LIN {X 0,Y 446.429,Z 349.503,A -85,B 0,C 180,E1 -8772.605,E2 -8772.605} C_VEL
LIN {X 0,Y 446.451,Z 349.5,A -85,B 0,C 180,E1 -8775.104,E2 -8775.104} C_VEL
LIN {X 0,Y 446.419,Z 349.505,A -85,B 0,C 180,E1 -8778.608,E2 -8778.608} C_VEL
LIN {X 0,Y 446.424,Z 349.503,A -85,B 0,C 180,E1 -8780.971,E2 -8780.971} C_VEL
LIN {X 0,Y 446.418,Z 349.505,A -85,B 0,C 180,E1 -8784.374,E2 -8784.374} C_VEL
LIN {X 0,Y 446.458,Z 349.655,A -85,B 0,C 180,E1 -8787.173,E2 -8787.173} C_VEL
LIN {X 0,Y 448.989,Z 357.621,A -85,B 0,C 180,E1 -8789.419,E2 -8789.419} C_VEL
